C09015=1043.792,433.131,-138.600,175.491,44.902,159.085
C09016=1043.804,433.376,-138.650,175.504,44.911,159.089
C09017=1043.815,433.620,-138.700,175.518,44.920,159.093
C09018=1043.827,433.865,-138.751,175.531,44.929,159.097
C09019=1043.838,434.091,-138.798,175.543,44.937,159.100
C09020=1043.848,434.319,-138.844,175.556,44.945,159.104
C09021=1043.860,434.545,-138.891,175.568,44.954,159.108
C09022=1043.870,434.771,-138.938,175.581,44.962,159.111
C09023=1043.881,434.997,-138.985,175.594,44.970,159.115
C09024=1043.892,435.223,-139.032,175.606,44.979,159.118
C09025=1043.903,435.450,-139.079,175.619,44.987,159.122
C09026=1043.914,435.676,-139.126,175.632,44.995,159.126
C09027=1043.926,435.921,-139.177,175.646,45.005,159.130
C09028=1043.938,436.166,-139.228,175.660,45.013,159.134
C09029=1043.949,436.409,-139.279,175.674,45.023,159.138
C09030=1043.961,436.654,-139.330,175.687,45.032,159.142
C09031=1043.973,436.898,-139.382,175.702,45.041,159.146
C09032=1043.985,437.143,-139.433,175.715,45.050,159.150
C09033=1043.997,437.388,-139.485,175.730,45.059,159.154
C09034=1044.010,437.632,-139.535,175.743,45.069,159.158
C09035=1044.021,437.876,-139.587,175.758,45.078,159.162
C09036=1044.033,438.121,-139.638,175.773,45.087,159.166
C09037=1044.046,438.365,-139.690,175.787,45.097,159.170
C09038=1044.057,438.609,-139.742,175.801,45.106,159.174
C09039=1044.069,438.854,-139.793,175.815,45.116,159.179
C09040=1044.081,439.098,-139.845,175.830,45.125,159.183
C09041=1044.093,439.342,-139.897,175.845,45.135,159.187
C09042=1044.106,439.587,-139.949,175.860,45.144,159.191
C09043=1044.118,439.831,-140.001,175.874,45.154,159.196
C09044=1044.130,440.075,-140.053,175.888,45.163,159.200
C09045=1044.142,440.319,-140.105,175.903,45.173,159.204
C09046=1044.155,440.564,-140.157,175.918,45.183,159.208
C09047=1044.167,440.808,-140.209,175.933,45.192,159.213
C09048=1044.179,441.052,-140.261,175.948,45.202,159.217
C09049=1044.192,441.297,-140.313,175.963,45.212,159.222
C09050=1044.204,441.540,-140.365,175.978,45.221,159.226
C09051=1044.216,441.784,-140.418,175.993,45.231,159.230
C09052=1044.230,442.028,-140.471,176.009,45.241,159.235
C09053=1044.242,442.272,-140.523,176.024,45.251,159.239
C09054=1044.255,442.517,-140.575,176.039,45.261,159.244
C09055=1044.267,442.761,-140.627,176.054,45.271,159.248
C09056=1044.279,443.005,-140.681,176.070,45.280,159.253
C09057=1044.292,443.249,-140.734,176.086,45.291,159.257
C09058=1044.304,443.493,-140.787,176.101,45.301,159.262
C09059=1044.317,443.737,-140.839,176.116,45.311,159.266
C09060=1044.330,443.981,-140.892,176.133,45.321,159.271
C09061=1044.343,444.225,-140.945,176.148,45.331,159.275
C09062=1044.355,444.469,-140.998,176.164,45.341,159.280
C09063=1044.368,444.712,-141.050,176.180,45.351,159.285
C09064=1044.381,444.956,-141.104,176.196,45.361,159.289
C09065=1044.394,445.199,-141.157,176.212,45.371,159.294
C09066=1044.408,445.443,-141.210,176.228,45.382,159.299
C09067=1044.421,445.686,-141.262,176.244,45.392,159.303
C09068=1044.436,445.929,-141.313,176.260,45.401,159.308
C09069=1044.451,446.173,-141.365,176.277,45.411,159.312
C09070=1044.467,446.417,-141.415,176.293,45.420,159.317
C09071=1044.483,446.661,-141.466,176.309,45.430,159.321
C09072=1044.500,446.904,-141.516,176.325,45.439,159.326
C09073=1044.518,447.148,-141.565,176.343,45.449,159.331
C09074=1044.536,447.393,-141.614,176.359,45.458,159.335
C09075=1044.555,447.637,-141.662,176.376,45.467,159.339
C09076=1044.575,447.881,-141.710,176.392,45.476,159.344
C09077=1044.595,448.126,-141.756,176.409,45.485,159.348
C09078=1044.616,448.370,-141.804,176.426,45.493,159.353
C09079=1044.635,448.593,-141.846,176.442,45.501,159.357
C09080=1044.656,448.816,-141.888,176.457,45.509,159.361
C09081=1044.676,449.038,-141.929,176.473,45.517,159.365
C09082=1044.697,449.261,-141.970,176.489,45.524,159.368
C09083=1044.719,449.485,-142.011,176.505,45.531,159.372
C09084=1044.740,449.707,-142.051,176.520,45.539,159.376
C09085=1044.763,449.931,-142.090,176.537,45.546,159.380
C09086=1044.787,450.153,-142.130,176.553,45.553,159.384
C09087=1044.813,450.399,-142.172,176.569,45.561,159.388
C09088=1044.839,450.644,-142.215,176.588,45.568,159.392
C09089=1044.867,450.890,-142.256,176.606,45.576,159.397
C09090=1044.894,451.135,-142.298,176.623,45.583,159.401
C09091=1044.591,451.173,-142.608,176.625,45.666,159.425
C09092=1044.562,450.927,-142.567,176.608,45.658,159.421
C09093=1044.535,450.683,-142.525,176.589,45.651,159.417
C09094=1044.508,450.437,-142.483,176.571,45.644,159.413
C09095=1044.482,450.192,-142.441,176.554,45.636,159.409
C09096=1044.460,449.977,-142.403,176.539,45.629,159.405
C09097=1044.438,449.762,-142.365,176.523,45.622,159.401
C09098=1044.416,449.547,-142.327,176.507,45.615,159.397
C09099=1044.395,449.333,-142.287,176.492,45.608,159.394
C09100=1044.374,449.118,-142.248,176.477,45.601,159.390
C09101=1044.354,448.903,-142.208,176.462,45.594,159.386
C09102=1044.335,448.689,-142.168,176.447,45.586,159.382
C09103=1044.316,448.474,-142.127,176.432,45.580,159.379
C09104=1044.294,448.229,-142.081,176.415,45.571,159.374
C09105=1044.274,447.985,-142.034,176.397,45.562,159.370
C09106=1044.254,447.740,-141.987,176.381,45.554,159.365
C09107=1044.235,447.496,-141.939,176.364,45.544,159.361
C09108=1044.215,447.252,-141.890,176.347,45.535,159.356
C09109=1044.198,447.008,-141.841,176.331,45.526,159.352
C09110=1044.181,446.764,-141.791,176.314,45.517,159.347
C09111=1044.164,446.521,-141.742,176.297,45.508,159.343
C09112=1044.147,446.276,-141.691,176.281,45.498,159.338
C09113=1044.132,446.032,-141.640,176.265,45.489,159.334
C09114=1044.117,445.789,-141.589,176.248,45.479,159.329
C09115=1044.103,445.546,-141.537,176.232,45.469,159.325
C09116=1044.089,445.302,-141.485,176.216,45.459,159.320
C09117=1044.076,445.059,-141.431,176.200,45.449,159.315
C09118=1044.063,444.816,-141.378,176.183,45.439,159.311
C09119=1044.050,444.573,-141.326,176.168,45.429,159.306
C09120=1044.037,444.329,-141.273,176.152,45.419,159.301
C09121=1044.025,444.085,-141.219,176.136,45.409,159.297
C09122=1044.012,443.841,-141.167,176.121,45.399,159.292
C09123=1043.999,443.597,-141.114,176.104,45.389,159.288
C09124=1043.986,443.353,-141.061,176.089,45.379,159.283
C09125=1043.974,443.109,-141.008,176.074,45.369,159.278
C09126=1043.961,442.865,-140.955,176.058,45.360,159.274
C09127=1043.949,442.621,-140.903,176.042,45.349,159.269
C09128=1043.936,442.376,-140.851,176.027,45.339,159.265
C09129=1043.923,442.133,-140.798,176.012,45.330,159.261
C09130=1043.910,441.888,-140.745,175.997,45.320,159.256
C09131=1043.898,441.645,-140.693,175.982,45.310,159.252
C09132=1043.886,441.400,-140.640,175.966,45.300,159.247
C09133=1043.874,441.156,-140.588,175.951,45.290,159.243
C09134=1043.861,440.911,-140.535,175.936,45.281,159.239
C09135=1043.849,440.667,-140.483,175.921,45.271,159.234
C09136=1043.837,440.423,-140.431,175.906,45.262,159.230
C09137=1043.824,440.179,-140.379,175.891,45.252,159.226
C09138=1043.812,439.935,-140.328,175.876,45.243,159.221
C09139=1043.799,439.691,-140.276,175.861,45.233,159.217
C09140=1043.787,439.447,-140.224,175.846,45.224,159.213
C09141=1043.775,439.202,-140.172,175.832,45.215,159.209
C09142=1043.762,438.958,-140.120,175.818,45.205,159.204
C09143=1043.751,438.713,-140.068,175.803,45.195,159.200
C09144=1043.738,438.469,-140.016,175.788,45.186,159.196
C09145=1043.727,438.225,-139.965,175.773,45.177,159.192
C09146=1043.715,437.980,-139.913,175.760,45.168,159.188
C09147=1043.702,437.736,-139.861,175.745,45.158,159.184
C09148=1043.691,437.492,-139.810,175.731,45.149,159.179
C09149=1043.679,437.247,-139.759,175.717,45.140,159.175
C09150=1043.666,437.003,-139.708,175.702,45.131,159.171
C09151=1043.654,436.759,-139.656,175.688,45.121,159.167
C09152=1043.642,436.514,-139.605,175.675,45.112,159.163
C09153=1043.631,436.270,-139.554,175.660,45.103,159.159
C09154=1043.619,436.025,-139.503,175.647,45.094,159.155
C09155=1043.608,435.781,-139.452,175.633,45.085,159.151
C09156=1043.596,435.554,-139.405,175.619,45.077,159.148
C09157=1043.585,435.326,-139.358,175.607,45.068,159.144
C09158=1043.574,435.099,-139.310,175.594,45.060,159.140
C09159=1043.562,434.872,-139.263,175.581,45.052,159.137
C09160=1043.552,434.645,-139.216,175.568,45.044,159.133
C09161=1043.541,434.417,-139.169,175.556,45.035,159.129
C09162=1043.530,434.190,-139.122,175.543,45.027,159.126
C09163=1043.519,433.963,-139.075,175.530,45.019,159.122
C09164=1043.508,433.718,-139.024,175.517,45.010,159.118
C09165=1043.495,433.473,-138.974,175.504,45.001,159.115
C09166=1043.484,433.229,-138.923,175.491,44.993,159.111
C09167=1043.472,432.984,-138.873,175.477,44.984,159.107
C09168=1043.461,432.740,-138.823,175.464,44.975,159.103
C09169=1043.449,432.495,-138.772,175.451,44.967,159.099
C09170=1043.438,432.250,-138.722,175.438,44.958,159.096
C09171=1043.427,432.006,-138.672,175.425,44.949,159.092
C09172=1043.414,431.761,-138.622,175.412,44.941,159.088
C09173=1043.404,431.516,-138.572,175.399,44.932,159.084
C09174=1043.392,431.271,-138.522,175.386,44.924,159.081
C09175=1043.380,431.027,-138.472,175.372,44.915,159.077
C09176=1043.370,430.782,-138.422,175.359,44.907,159.073
C09177=1043.358,430.538,-138.372,175.347,44.898,159.070
C09178=1043.346,430.293,-138.322,175.334,44.890,159.066
C09179=1043.336,430.047,-138.272,175.322,44.881,159.063
C09180=1043.324,429.803,-138.222,175.309,44.873,159.059
C09181=1043.313,429.558,-138.173,175.296,44.864,159.055
C09182=1043.302,429.314,-138.124,175.283,44.856,159.052
C09183=1043.291,429.069,-138.073,175.271,44.848,159.048
C09184=1043.280,428.823,-138.024,175.258,44.840,159.045
C09185=1043.268,428.579,-137.974,175.245,44.831,159.041
C09186=1043.257,428.334,-137.925,175.234,44.823,159.038
C09187=1043.246,428.089,-137.876,175.221,44.815,159.034
C09188=1043.235,427.844,-137.827,175.208,44.807,159.031
C09189=1043.224,427.599,-137.777,175.196,44.799,159.027
C09190=1043.213,427.354,-137.728,175.184,44.791,159.024
C09191=1043.201,427.110,-137.679,175.172,44.782,159.020
C09192=1043.191,426.865,-137.630,175.159,44.774,159.017
C09193=1043.180,426.619,-137.581,175.148,44.766,159.014
C09194=1043.168,426.374,-137.532,175.135,44.758,159.010
C09195=1043.158,426.129,-137.483,175.123,44.750,159.007
C09196=1043.147,425.885,-137.435,175.111,44.742,159.003
C09197=1043.136,425.640,-137.386,175.099,44.734,159.000
C09198=1043.125,425.395,-137.336,175.087,44.726,158.997
C09199=1043.114,425.150,-137.288,175.075,44.719,158.993
C09200=1043.103,424.906,-137.239,175.063,44.710,158.990
C09201=1043.092,424.660,-137.191,175.051,44.703,158.987
C09202=1043.082,424.414,-137.142,175.040,44.695,158.983
C09203=1043.070,424.169,-137.094,175.028,44.687,158.980
C09204=1043.060,423.925,-137.045,175.017,44.679,158.977
C09205=1043.049,423.680,-136.997,175.004,44.671,158.974
C09206=1043.037,423.434,-136.948,174.993,44.664,158.970
C09207=1043.027,423.190,-136.901,174.981,44.656,158.967
C09208=1043.016,422.944,-136.852,174.970,44.648,158.964
C09209=1043.005,422.700,-136.804,174.959,44.641,158.961
C09210=1042.995,422.454,-136.755,174.946,44.633,158.957
C09211=1042.984,422.209,-136.707,174.935,44.626,158.954
C09212=1042.974,421.963,-136.660,174.924,44.618,158.951
C09213=1042.963,421.718,-136.612,174.913,44.610,158.948
C09214=1042.952,421.473,-136.564,174.901,44.602,158.945
C09215=1042.942,421.229,-136.516,174.890,44.595,158.942
C09216=1042.933,421.011,-136.474,174.881,44.589,158.939
C09217=1042.922,420.793,-136.431,174.870,44.582,158.936
C09218=1042.913,420.575,-136.388,174.860,44.575,158.934
C09219=1042.904,420.358,-136.346,174.850,44.568,158.931
C09220=1042.894,420.140,-136.304,174.841,44.562,158.928
C09221=1042.885,419.922,-136.261,174.831,44.555,158.925
C09222=1042.876,419.704,-136.219,174.821,44.549,158.923
C09223=1042.866,419.487,-136.177,174.811,44.542,158.920
C09224=1042.856,419.242,-136.129,174.800,44.535,158.917
C09225=1042.846,418.997,-136.082,174.790,44.528,158.914
C09226=1042.835,418.752,-136.034,174.778,44.520,158.911
C09227=1042.825,418.507,-135.987,174.767,44.513,158.908
C09228=1042.815,418.260,-135.939,174.756,44.506,158.905
C09229=1042.804,418.015,-135.892,174.745,44.499,158.902
C09230=1042.794,417.770,-135.845,174.735,44.491,158.899
C09231=1042.784,417.525,-135.798,174.724,44.484,158.896
C09232=1042.774,417.279,-135.751,174.713,44.477,158.893
C09233=1042.764,417.034,-135.703,174.703,44.470,158.890
C09234=1042.752,416.789,-135.656,174.692,44.462,158.887
C09235=1042.742,416.543,-135.609,174.682,44.456,158.884
C09236=1042.732,416.297,-135.563,174.671,44.449,158.881
C09237=1042.722,416.052,-135.515,174.661,44.442,158.879
C09238=1042.712,415.807,-135.468,174.650,44.434,158.876
C09239=1042.701,415.561,-135.422,174.639,44.427,158.873
C09240=1042.691,415.317,-135.375,174.629,44.420,158.870
C09241=1042.681,415.071,-135.328,174.618,44.413,158.867
C09242=1042.671,414.825,-135.282,174.609,44.406,158.864
C09243=1042.660,414.580,-135.235,174.598,44.399,158.861
C09244=1042.650,414.335,-135.189,174.588,44.393,158.859
C09245=1042.640,414.089,-135.141,174.577,44.386,158.856
C09246=1042.630,413.843,-135.095,174.568,44.379,158.853
C09247=1042.620,413.598,-135.049,174.557,44.372,158.850
C09248=1042.610,413.353,-135.002,174.547,44.365,158.848
C09249=1042.600,413.107,-134.956,174.537,44.358,158.845
C09250=1042.590,412.861,-134.909,174.527,44.351,158.842
C09251=1042.580,412.616,-134.864,174.516,44.345,158.839
C09252=1042.571,412.371,-134.817,174.506,44.338,158.836
C09253=1042.560,412.125,-134.770,174.497,44.331,158.834
C09254=1042.551,411.880,-134.724,174.486,44.325,158.831
C09255=1042.541,411.634,-134.679,174.477,44.318,158.828
C09256=1042.530,411.388,-134.633,174.466,44.311,158.826
C09257=1042.521,411.143,-134.586,174.457,44.305,158.823
C09258=1042.510,410.897,-134.541,174.447,44.298,158.820
C09259=1042.500,410.652,-134.494,174.436,44.292,158.818
C09260=1042.490,410.407,-134.449,174.427,44.285,158.815
C09261=1042.481,410.160,-134.403,174.417,44.278,158.813
C09262=1042.471,409.915,-134.357,174.408,44.272,158.810
C09263=1042.460,409.670,-134.311,174.397,44.265,158.807
C09264=1042.451,409.424,-134.266,174.388,44.259,158.805
C09265=1042.440,409.178,-134.220,174.378,44.252,158.802
C09266=1042.431,408.932,-134.175,174.369,44.246,158.800
C09267=1042.421,408.688,-134.129,174.360,44.239,158.797
C09268=1042.412,408.441,-134.083,174.349,44.233,158.794
C09269=1042.402,408.196,-134.038,174.340,44.227,158.792
C09270=1042.392,407.950,-133.993,174.330,44.220,158.789
C09271=1042.383,407.704,-133.947,174.321,44.214,158.787
C09272=1042.373,407.459,-133.902,174.312,44.207,158.784
C09273=1042.364,407.213,-133.856,174.302,44.201,158.782
C09274=1042.353,406.967,-133.811,174.293,44.195,158.779
C09275=1042.344,406.722,-133.766,174.284,44.189,158.777
C09276=1042.336,406.508,-133.727,174.275,44.183,158.774
C09277=1042.327,406.295,-133.687,174.267,44.178,158.772
C09278=1042.319,406.081,-133.648,174.259,44.172,158.770
C09279=1042.310,405.867,-133.608,174.251,44.167,158.768
C09280=1042.302,405.654,-133.569,174.242,44.161,158.766
C09281=1042.293,405.440,-133.530,174.235,44.156,158.764
C09282=1042.285,405.227,-133.490,174.227,44.150,158.762
C09283=1042.278,405.013,-133.452,174.219,44.145,158.759
C09284=1042.268,404.767,-133.407,174.210,44.139,158.757
C09285=1042.258,404.522,-133.362,174.200,44.133,158.755
C09286=1042.249,404.276,-133.317,174.191,44.127,158.752
C09287=1042.240,404.030,-133.272,174.182,44.121,158.750
C09288=1042.230,403.784,-133.228,174.173,44.115,158.747
C09289=1042.221,403.538,-133.182,174.164,44.109,158.745
C09290=1042.211,403.292,-133.137,174.155,44.102,158.743
C09291=1042.201,403.046,-133.093,174.146,44.097,158.740
C09292=1042.192,402.801,-133.048,174.137,44.090,158.738
C09293=1042.183,402.555,-133.003,174.128,44.084,158.735
C09294=1042.174,402.309,-132.959,174.119,44.079,158.733
C09295=1042.164,402.064,-132.914,174.110,44.073,158.731
C09296=1042.155,401.818,-132.870,174.102,44.067,158.729
C09297=1042.145,401.572,-132.826,174.093,44.061,158.726
C09298=1042.136,401.326,-132.781,174.084,44.055,158.724
C09299=1042.126,401.080,-132.737,174.075,44.049,158.721
C09300=1042.118,400.834,-132.693,174.067,44.043,158.719
C09301=1042.108,400.589,-132.648,174.058,44.037,158.717
C09302=1042.099,400.343,-132.604,174.049,44.031,158.715
C09303=1042.090,400.096,-132.560,174.040,44.026,158.712
C09304=1042.080,399.851,-132.516,174.032,44.020,158.710
C09305=1042.071,399.605,-132.472,174.023,44.014,158.708
C09306=1042.061,399.359,-132.428,174.014,44.009,158.706
C09307=1042.052,399.113,-132.384,174.006,44.003,158.703
C09308=1042.043,398.867,-132.340,173.997,43.997,158.701
C09309=1042.034,398.621,-132.296,173.988,43.992,158.699
C09310=1042.024,398.375,-132.252,173.980,43.986,158.697
C09311=1042.016,398.130,-132.208,173.971,43.980,158.695
C09312=1042.006,397.884,-132.164,173.962,43.974,158.692
C09313=1041.997,397.638,-132.121,173.954,43.969,158.690
C09314=1041.988,397.392,-132.076,173.945,43.963,158.688
C09315=1041.979,397.147,-132.033,173.938,43.957,158.686
C09316=1041.969,396.900,-131.990,173.929,43.952,158.684
C09317=1041.960,396.655,-131.946,173.921,43.946,158.681
C09318=1041.951,396.409,-131.902,173.912,43.941,158.679
C09319=1041.943,396.163,-131.859,173.904,43.935,158.677
C09320=1041.933,395.916,-131.815,173.895,43.930,158.675
C09321=1041.924,395.671,-131.771,173.888,43.924,158.673
C09322=1041.915,395.424,-131.728,173.879,43.919,158.671
C09323=1041.906,395.179,-131.685,173.871,43.913,158.669
C09324=1041.897,394.933,-131.642,173.862,43.908,158.666
C09325=1041.888,394.686,-131.598,173.855,43.902,158.664
C09326=1041.879,394.441,-131.554,173.846,43.897,158.662
C09327=1041.869,394.194,-131.512,173.838,43.892,158.660
C09328=1041.861,393.948,-131.469,173.829,43.886,158.658
C09329=1041.852,393.703,-131.425,173.822,43.881,158.656
C09330=1041.842,393.456,-131.382,173.813,43.875,158.654
C09331=1041.834,393.210,-131.339,173.805,43.870,158.652
C09332=1041.825,392.964,-131.296,173.798,43.865,158.650
C09333=1041.816,392.719,-131.253,173.789,43.860,158.648
C09334=1041.807,392.472,-131.209,173.781,43.854,158.646
C09335=1041.798,392.226,-131.166,173.774,43.849,158.644
C09336=1041.783,391.818,-131.096,173.760,43.840,158.640
C09337=1041.769,391.411,-131.025,173.747,43.831,158.637
C09338=1041.754,391.003,-130.954,173.733,43.823,158.634
C09339=1041.739,390.595,-130.883,173.720,43.814,158.630
C09340=1041.731,390.349,-130.840,173.713,43.809,158.628
C09341=1041.722,390.103,-130.798,173.705,43.804,158.627
C09342=1041.713,389.857,-130.755,173.697,43.799,158.624
C09343=1041.704,389.610,-130.713,173.689,43.794,158.622
C09344=1041.695,389.364,-130.670,173.681,43.789,158.621
C09345=1041.686,389.119,-130.627,173.674,43.784,158.619
C09346=1041.678,388.872,-130.585,173.666,43.778,158.617
C09347=1041.668,388.626,-130.543,173.658,43.774,158.615
C09348=1041.660,388.379,-130.500,173.650,43.768,158.613
C09349=1041.651,388.134,-130.458,173.643,43.764,158.611
C09350=1041.643,387.887,-130.416,173.635,43.759,158.609
C09351=1041.634,387.641,-130.373,173.628,43.753,158.607
C09352=1041.625,387.395,-130.331,173.619,43.749,158.605
C09353=1041.616,387.148,-130.289,173.612,43.744,158.603
C09354=1041.607,386.902,-130.247,173.604,43.739,158.601
C09355=1041.598,386.656,-130.205,173.597,43.734,158.600
C09356=1041.589,386.410,-130.163,173.590,43.729,158.598
C09357=1041.581,386.164,-130.120,173.582,43.724,158.596
C09358=1041.572,385.918,-130.079,173.575,43.720,158.594
C09359=1041.564,385.672,-130.037,173.566,43.714,158.592
C09360=1041.555,385.425,-129.995,173.559,43.710,158.590
C09361=1041.546,385.179,-129.953,173.552,43.705,158.588
C09362=1041.537,384.932,-129.911,173.544,43.700,158.587
C09363=1041.529,384.686,-129.870,173.537,43.695,158.585
C09364=1041.520,384.440,-129.828,173.530,43.690,158.583
C09365=1041.512,384.194,-129.786,173.522,43.686,158.581
C09366=1041.503,383.947,-129.744,173.515,43.681,158.579
C09367=1041.494,383.701,-129.703,173.508,43.677,158.578
C09368=1041.486,383.455,-129.661,173.500,43.672,158.576
C09369=1041.477,383.209,-129.620,173.493,43.667,158.574
C09370=1041.469,382.962,-129.577,173.486,43.662,158.572
C09371=1041.460,382.716,-129.536,173.478,43.657,158.570
C09372=1041.452,382.469,-129.495,173.471,43.652,158.568
C09373=1041.443,382.223,-129.453,173.464,43.648,158.567
C09374=1041.435,381.977,-129.411,173.456,43.643,158.565
C09375=1041.426,381.731,-129.369,173.449,43.639,158.563
C09376=1041.418,381.484,-129.328,173.442,43.634,158.561
C09377=1041.409,381.238,-129.287,173.435,43.630,158.560
C09378=1041.400,380.992,-129.245,173.427,43.625,158.558
C09379=1041.393,380.745,-129.204,173.421,43.620,158.556
C09380=1041.384,380.499,-129.162,173.414,43.615,158.554
C09381=1041.376,380.253,-129.122,173.407,43.611,158.553
C09382=1041.367,380.006,-129.080,173.399,43.606,158.551
C09383=1041.359,379.760,-129.039,173.392,43.602,158.549
C09384=1041.347,379.392,-128.977,173.382,43.595,158.547
C09385=1041.334,379.025,-128.916,173.372,43.588,158.544
C09386=1041.322,378.657,-128.854,173.360,43.582,158.542
C09387=1041.309,378.290,-128.794,173.350,43.575,158.539
C09388=1041.300,378.043,-128.753,173.343,43.571,158.537
C09389=1041.292,377.797,-128.712,173.337,43.566,158.536
C09390=1041.284,377.551,-128.672,173.330,43.562,158.534
C09391=1041.275,377.304,-128.630,173.323,43.558,158.533
C09392=1041.267,377.051,-128.589,173.315,43.553,158.531
C09393=1041.259,376.798,-128.547,173.308,43.549,158.529
C09394=1041.250,376.546,-128.505,173.301,43.544,158.527
C09395=1041.241,376.293,-128.463,173.294,43.540,158.526
C09396=1041.233,376.046,-128.423,173.288,43.535,158.524
C09397=1041.224,375.799,-128.382,173.281,43.531,158.523
C09398=1041.216,375.553,-128.341,173.274,43.527,158.521
C09399=1041.208,375.307,-128.300,173.267,43.523,158.519
C09400=1041.200,375.060,-128.260,173.261,43.518,158.518
C09401=1041.192,374.813,-128.219,173.254,43.514,158.516
C09402=1041.183,374.567,-128.179,173.246,43.510,158.514
C09403=1041.175,374.321,-128.139,173.240,43.505,158.513
C09404=1041.167,374.074,-128.098,173.233,43.502,158.511
C09405=1041.159,373.827,-128.058,173.226,43.497,158.510
C09406=1041.151,373.581,-128.017,173.220,43.493,158.508
C09407=1041.143,373.334,-127.977,173.213,43.488,158.506
C09408=1041.134,373.088,-127.937,173.206,43.485,158.505
C09409=1041.126,372.841,-127.897,173.200,43.480,158.503
C09410=1041.117,372.594,-127.856,173.193,43.476,158.502
C09411=1041.110,372.347,-127.816,173.186,43.472,158.500
C09412=1041.102,372.101,-127.775,173.180,43.468,158.499
C09413=1041.094,371.854,-127.735,173.173,43.463,158.497
C09414=1041.085,371.608,-127.695,173.167,43.459,158.496
C09415=1041.077,371.361,-127.655,173.160,43.455,158.494
C09416=1041.069,371.115,-127.615,173.153,43.451,158.492
C09417=1041.062,370.868,-127.575,173.147,43.447,158.491
C09418=1041.054,370.622,-127.534,173.141,43.443,158.489
C09419=1041.045,370.375,-127.495,173.134,43.439,158.488
C09420=1041.038,370.128,-127.455,173.128,43.435,158.486
C09421=1041.029,369.882,-127.415,173.122,43.431,158.485
C09422=1041.021,369.636,-127.375,173.115,43.427,158.483
C09423=1041.013,369.389,-127.335,173.108,43.423,158.482
C09424=1041.004,369.141,-127.295,173.102,43.419,158.480
C09425=1040.996,368.895,-127.256,173.095,43.415,158.479
C09426=1040.988,368.648,-127.216,173.089,43.411,158.477
C09427=1040.980,368.403,-127.176,173.082,43.408,158.476
C09428=1040.972,368.156,-127.136,173.076,43.403,158.474
C09429=1040.964,367.909,-127.097,173.070,43.399,158.473
C09430=1040.956,367.662,-127.057,173.064,43.395,158.471
C09431=1040.948,367.416,-127.018,173.057,43.392,158.470
C09432=1040.940,367.169,-126.978,173.051,43.388,158.469
C09433=1040.931,366.922,-126.939,173.044,43.384,158.467
C09434=1040.924,366.675,-126.899,173.038,43.380,158.466
C09435=1040.916,366.428,-126.860,173.033,43.376,158.464
C09436=1040.908,366.181,-126.820,173.026,43.372,158.463
C09437=1040.899,365.934,-126.781,173.020,43.368,158.461
C09438=1040.892,365.688,-126.741,173.013,43.365,158.460
C09439=1040.884,365.442,-126.702,173.007,43.361,158.458
C09440=1040.876,365.194,-126.663,173.000,43.357,158.457
C09441=1040.868,364.948,-126.623,172.995,43.353,158.456
C09442=1040.860,364.701,-126.583,172.989,43.350,158.454
C09443=1040.852,364.455,-126.545,172.982,43.346,158.453
C09444=1040.844,364.208,-126.506,172.976,43.342,158.451
C09445=1040.836,363.961,-126.466,172.970,43.338,158.450
C09446=1040.828,363.714,-126.427,172.964,43.334,158.448
C09447=1040.821,363.467,-126.388,172.958,43.331,158.447
C09448=1040.809,363.113,-126.331,172.950,43.325,158.445
C09449=1040.799,362.759,-126.275,172.940,43.320,158.443
C09450=1040.788,362.405,-126.219,172.932,43.315,158.441
C09451=1040.776,362.051,-126.164,172.923,43.309,158.439
C09452=1040.769,361.804,-126.124,172.917,43.305,158.438
C09453=1040.760,361.557,-126.085,172.911,43.302,158.437
C09454=1040.753,361.311,-126.047,172.905,43.298,158.435
C09455=1040.744,361.064,-126.008,172.899,43.295,158.434
C09456=1040.736,360.816,-125.970,172.892,43.291,158.432
C09457=1040.729,360.570,-125.930,172.887,43.288,158.431
C09458=1040.721,360.323,-125.891,172.881,43.284,158.430
C09459=1040.713,360.076,-125.853,172.875,43.280,158.428
C09460=1040.705,359.829,-125.815,172.869,43.277,158.427
C09461=1040.697,359.582,-125.776,172.863,43.273,158.426
C09462=1040.689,359.336,-125.737,172.857,43.270,158.425
C09463=1040.682,359.089,-125.698,172.851,43.266,158.423
C09464=1040.674,358.842,-125.660,172.845,43.263,158.422
C09465=1040.666,358.595,-125.621,172.840,43.259,158.421
C09466=1040.659,358.348,-125.583,172.834,43.256,158.419
C09467=1040.650,358.101,-125.544,172.828,43.252,158.418
C09468=1040.643,357.855,-125.506,172.822,43.249,158.417
C09469=1040.635,357.607,-125.467,172.816,43.245,158.415
C09470=1040.627,357.361,-125.429,172.810,43.242,158.414
C09471=1040.620,357.113,-125.390,172.805,43.238,158.413
C09472=1040.612,356.867,-125.352,172.799,43.234,158.411
C09473=1040.604,356.619,-125.314,172.792,43.231,158.410
C09474=1040.597,356.372,-125.275,172.787,43.228,158.409
C09475=1040.589,356.126,-125.237,172.781,43.224,158.408
C09476=1040.581,355.879,-125.199,172.776,43.221,158.406
C09477=1040.574,355.632,-125.160,172.770,43.218,158.405
C09478=1040.566,355.384,-125.122,172.765,43.214,158.404
C09479=1040.558,355.138,-125.084,172.758,43.211,158.403
C09480=1040.549,354.891,-125.046,172.752,43.208,158.401
C09481=1040.542,354.644,-125.009,172.747,43.204,158.400
C09482=1040.535,354.397,-124.970,172.741,43.201,158.399
C09483=1040.527,354.149,-124.932,172.736,43.198,158.398
C09484=1040.519,353.903,-124.894,172.730,43.194,158.396
C09485=1040.512,353.656,-124.856,172.725,43.191,158.395
C09486=1040.504,353.409,-124.818,172.718,43.188,158.394
C09487=1040.496,353.162,-124.780,172.713,43.184,158.393
C09488=1040.489,352.915,-124.742,172.707,43.181,158.391
C09489=1040.481,352.668,-124.704,172.702,43.178,158.390
C09490=1040.474,352.421,-124.666,172.696,43.175,158.389
C09491=1040.466,352.174,-124.629,172.691,43.171,158.388
C09492=1040.458,351.927,-124.591,172.685,43.168,158.387
C09493=1040.451,351.680,-124.553,172.680,43.165,158.385
C09494=1040.443,351.433,-124.515,172.674,43.162,158.384
C09495=1040.435,351.186,-124.477,172.669,43.158,158.383
C09496=1040.428,350.939,-124.440,172.663,43.155,158.382
C09497=1040.421,350.692,-124.402,172.658,43.152,158.381
C09498=1040.413,350.445,-124.364,172.652,43.149,158.379
C09499=1040.405,350.198,-124.327,172.647,43.146,158.378
C09500=1040.397,349.950,-124.289,172.641,43.142,158.377
C09501=1040.390,349.703,-124.252,172.636,43.139,158.376
C09502=1040.383,349.457,-124.213,172.630,43.136,158.375
C09503=1040.375,349.210,-124.177,172.625,43.133,158.373
C09504=1040.364,348.861,-124.124,172.617,43.128,158.372
C09505=1040.354,348.514,-124.071,172.609,43.124,158.370
C09506=1040.342,348.165,-124.019,172.602,43.120,158.369
C09507=1040.332,347.817,-123.966,172.594,43.115,158.367
C09508=1040.324,347.570,-123.929,172.588,43.112,158.366
C09509=1040.317,347.323,-123.891,172.583,43.109,158.365
C09510=1040.310,347.076,-123.854,172.577,43.106,158.364
C09511=1040.302,346.829,-123.817,172.572,43.103,158.362
C09512=1040.295,346.581,-123.780,172.566,43.100,158.361
C09513=1040.288,346.334,-123.742,172.562,43.097,158.360
C09514=1040.280,346.087,-123.705,172.557,43.094,158.359
C09515=1040.273,345.840,-123.668,172.551,43.091,158.358
C09516=1040.265,345.594,-123.631,172.546,43.088,158.357
C09517=1040.258,345.346,-123.594,172.541,43.085,158.356
C09518=1040.250,345.099,-123.557,172.535,43.082,158.355
C09519=1040.242,344.852,-123.520,172.530,43.079,158.354
C09520=1040.235,344.605,-123.482,172.524,43.076,158.352
C09521=1040.228,344.357,-123.446,172.519,43.073,158.351
C09522=1040.220,344.110,-123.408,172.514,43.070,158.350
C09523=1040.212,343.863,-123.371,172.508,43.067,158.349
C09524=1040.205,343.616,-123.335,172.504,43.064,158.348
C09525=1040.197,343.369,-123.298,172.499,43.061,158.347
C09526=1040.190,343.121,-123.261,172.493,43.058,158.346
C09527=1040.183,342.875,-123.224,172.488,43.055,158.345
C09528=1040.176,342.627,-123.187,172.483,43.052,158.343
C09529=1040.168,342.380,-123.151,172.477,43.049,158.342
C09530=1040.161,342.132,-123.114,172.473,43.046,158.341
C09531=1040.153,341.886,-123.077,172.468,43.043,158.340
C09532=1040.146,341.638,-123.040,172.462,43.040,158.339
C09533=1040.138,341.391,-123.003,172.457,43.038,158.338
C09534=1040.131,341.144,-122.967,172.452,43.035,158.337
C09535=1040.124,340.897,-122.930,172.446,43.032,158.336
C09536=1040.116,340.650,-122.893,172.442,43.029,158.335
C09537=1040.109,340.402,-122.857,172.437,43.026,158.334
C09538=1040.102,340.155,-122.820,172.431,43.024,158.333
C09539=1040.095,339.908,-122.785,172.426,43.021,158.332
C09540=1040.087,339.661,-122.748,172.421,43.018,158.331
C09541=1040.079,339.414,-122.711,172.417,43.015,158.330
C09542=1040.072,339.166,-122.675,172.411,43.013,158.329
C09543=1040.064,338.918,-122.638,172.406,43.010,158.328
C09544=1040.057,338.672,-122.603,172.401,43.007,158.327
C09545=1040.049,338.425,-122.566,172.396,43.004,158.326
C09546=1040.042,338.177,-122.529,172.391,43.001,158.325
C09547=1040.035,337.930,-122.493,172.386,42.999,158.324
C09548=1040.028,337.683,-122.457,172.381,42.996,158.322
C09549=1040.021,337.435,-122.420,172.376,42.993,158.322
C09550=1040.014,337.188,-122.384,172.371,42.990,158.321
C09551=1040.006,336.941,-122.348,172.366,42.987,158.319
C09552=1039.998,336.693,-122.312,172.361,42.985,158.319
C09553=1039.992,336.446,-122.275,172.357,42.982,158.317
C09554=1039.984,336.199,-122.239,172.351,42.979,158.316
C09555=1039.977,335.951,-122.203,172.346,42.977,158.316
C09556=1039.969,335.705,-122.167,172.341,42.974,158.314
C09557=1039.962,335.457,-122.131,172.337,42.972,158.314
C09558=1039.955,335.210,-122.094,172.331,42.969,158.312
C09559=1039.948,334.962,-122.059,172.326,42.966,158.311
C09560=1039.937,334.611,-122.008,172.320,42.962,158.310
C09561=1039.927,334.259,-121.957,172.313,42.959,158.309
C09562=1039.917,333.907,-121.906,172.306,42.955,158.307
C09563=1039.907,333.555,-121.855,172.298,42.952,158.306
C09564=1039.899,333.308,-121.818,172.294,42.948,158.305
C09565=1039.892,333.061,-121.783,172.289,42.946,158.304
C09566=1039.885,332.813,-121.747,172.284,42.943,158.303
C09567=1039.877,332.566,-121.711,172.280,42.941,158.302
C09568=1039.869,332.319,-121.676,172.275,42.938,158.301
C09569=1039.862,332.072,-121.640,172.269,42.936,158.300
C09570=1039.855,331.824,-121.604,172.265,42.933,158.299
C09571=1039.848,331.577,-121.569,172.260,42.931,158.298
C09572=1039.840,331.330,-121.533,172.256,42.928,158.297
C09573=1039.833,331.082,-121.498,172.251,42.925,158.296
C09574=1039.826,330.835,-121.462,172.246,42.923,158.295
C09575=1039.819,330.587,-121.426,172.241,42.920,158.294
C09576=1039.812,330.341,-121.391,172.236,42.918,158.293
C09577=1039.804,330.093,-121.355,172.232,42.915,158.293
C09578=1039.797,329.846,-121.319,172.227,42.913,158.292
C09579=1039.790,329.598,-121.284,172.222,42.910,158.291
C09580=1039.783,329.350,-121.249,172.218,42.908,158.290
C09581=1039.776,329.104,-121.213,172.213,42.905,158.289
C09582=1039.769,328.856,-121.177,172.208,42.903,158.288
C09583=1039.762,328.608,-121.142,172.203,42.900,158.287
C09584=1039.754,328.361,-121.106,172.198,42.898,158.286
C09585=1039.747,328.114,-121.071,172.194,42.896,158.285
C09586=1039.740,327.866,-121.036,172.189,42.893,158.284
C09587=1039.732,327.619,-121.001,172.185,42.891,158.283
C09588=1039.725,327.371,-120.966,172.180,42.889,158.283
C09589=1039.717,327.123,-120.931,172.175,42.886,158.282
C09590=1039.710,326.876,-120.896,172.171,42.884,158.281
C09591=1039.703,326.629,-120.862,172.166,42.881,158.280
C09592=1039.695,326.382,-120.825,172.162,42.879,158.279
C09593=1039.688,326.135,-120.791,172.156,42.877,158.278
C09594=1039.681,325.887,-120.756,172.152,42.874,158.277
C09595=1039.674,325.639,-120.720,172.147,42.872,158.276
C09596=1039.666,325.392,-120.686,172.143,42.869,158.275
C09597=1039.659,325.145,-120.651,172.138,42.867,158.274
C09598=1039.652,324.898,-120.616,172.134,42.865,158.274
C09599=1039.645,324.649,-120.581,172.129,42.863,158.273
C09600=1039.637,324.402,-120.547,172.125,42.860,158.272
C09601=1039.630,324.155,-120.512,172.120,42.858,158.271
C09602=1039.623,323.908,-120.477,172.115,42.856,158.270
C09603=1039.616,323.659,-120.441,172.111,42.853,158.269
C09604=1039.608,323.412,-120.407,172.107,42.851,158.268
C09605=1039.601,323.165,-120.372,172.102,42.849,158.268
C09606=1039.594,322.918,-120.337,172.098,42.846,158.267
C09607=1039.587,322.670,-120.303,172.093,42.844,158.266
C09608=1039.580,322.422,-120.267,172.089,42.842,158.265
C09609=1039.572,322.175,-120.233,172.084,42.839,158.264
C09610=1039.566,321.928,-120.198,172.080,42.837,158.263
C09611=1039.558,321.680,-120.164,172.075,42.835,158.262
C09612=1039.552,321.432,-120.129,172.070,42.833,158.262
C09613=1039.544,321.185,-120.094,172.065,42.830,158.261
C09614=1039.538,320.937,-120.060,172.062,42.828,158.260
C09615=1039.530,320.690,-120.025,172.056,42.826,158.259
C09616=1039.520,320.333,-119.975,172.051,42.823,158.258
C09617=1039.509,319.977,-119.926,172.045,42.820,158.257
C09618=1039.499,319.621,-119.875,172.038,42.816,158.255
C09619=1039.489,319.264,-119.825,172.032,42.813,158.254
C09620=1039.482,319.017,-119.791,172.027,42.811,158.253
C09621=1039.475,318.769,-119.756,172.023,42.809,158.253
C09622=1039.468,318.522,-119.722,172.019,42.806,158.252
C09623=1039.461,318.274,-119.687,172.014,42.805,158.251
C09624=1039.454,318.027,-119.653,172.010,42.802,158.250
C09625=1039.447,317.779,-119.618,172.005,42.800,158.249
C09626=1039.440,317.532,-119.584,172.001,42.798,158.248
C09627=1039.433,317.284,-119.549,171.997,42.795,158.248
C09628=1039.426,317.036,-119.515,171.992,42.794,158.247
C09629=1039.420,316.788,-119.481,171.988,42.791,158.246
C09630=1039.413,316.542,-119.447,171.984,42.789,158.245
C09631=1039.406,316.294,-119.413,171.979,42.787,158.244
C09632=1039.399,316.047,-119.378,171.975,42.784,158.243
C09633=1039.392,315.799,-119.344,171.971,42.782,158.243
C09634=1039.385,315.551,-119.310,171.966,42.780,158.242
C09635=1039.378,315.304,-119.275,171.962,42.778,158.241
C09636=1039.371,315.056,-119.241,171.958,42.776,158.240
C09637=1039.364,314.809,-119.207,171.953,42.774,158.239
C09638=1039.358,314.562,-119.172,171.949,42.771,158.239
C09639=1039.351,314.314,-119.138,171.945,42.769,158.238
C09640=1039.344,314.066,-119.104,171.941,42.767,158.237
C09641=1039.337,313.819,-119.070,171.936,42.765,158.236
C09642=1039.330,313.571,-119.036,171.932,42.763,158.235
C09643=1039.324,313.324,-119.001,171.928,42.761,158.235
C09644=1039.316,313.077,-118.968,171.923,42.759,158.234
C09645=1039.310,312.829,-118.933,171.919,42.756,158.233
C09646=1039.303,312.581,-118.899,171.915,42.755,158.232
C09647=1039.297,312.334,-118.865,171.911,42.752,158.231
C09648=1039.290,312.086,-118.831,171.906,42.750,158.231
C09649=1039.282,311.838,-118.798,171.903,42.748,158.230
C09650=1039.275,311.591,-118.764,171.899,42.746,158.229
C09651=1039.268,311.343,-118.730,171.894,42.744,158.228
C09652=1039.261,311.095,-118.696,171.890,42.742,158.228
C09653=1039.253,310.849,-118.663,171.886,42.740,158.227
C09654=1039.246,310.601,-118.629,171.882,42.738,158.226
C09655=1039.239,310.353,-118.596,171.877,42.737,158.225
C09656=1039.232,310.105,-118.562,171.873,42.735,158.225
C09657=1039.225,309.857,-118.529,171.869,42.733,158.224
C09658=1039.218,309.610,-118.495,171.865,42.731,158.223
C09659=1039.211,309.363,-118.461,171.861,42.728,158.222
C09660=1039.203,309.115,-118.428,171.857,42.727,158.222
C09661=1039.196,308.867,-118.395,171.853,42.725,158.221
C09662=1039.190,308.620,-118.362,171.848,42.723,158.220
C09663=1039.183,308.373,-118.328,171.844,42.721,158.220
C09664=1039.176,308.124,-118.295,171.840,42.719,158.219
C09665=1039.168,307.877,-118.261,171.836,42.717,158.218
C09666=1039.161,307.630,-118.228,171.832,42.715,158.217
C09667=1039.154,307.382,-118.194,171.828,42.713,158.217
C09668=1039.147,307.134,-118.161,171.824,42.712,158.216
C09669=1039.140,306.887,-118.128,171.820,42.710,158.215
C09670=1039.134,306.639,-118.094,171.815,42.708,158.214
C09671=1039.126,306.391,-118.061,171.811,42.706,158.214
C09672=1039.116,306.040,-118.014,171.806,42.703,158.213
C09673=1039.106,305.688,-117.967,171.800,42.701,158.212
C09674=1039.097,305.336,-117.920,171.795,42.698,158.211
C09675=1039.087,304.985,-117.872,171.788,42.695,158.210
C09676=1039.080,304.737,-117.839,171.784,42.693,158.209
C09677=1039.072,304.490,-117.806,171.781,42.691,158.208
C09678=1039.065,304.241,-117.773,171.776,42.689,158.207
C09679=1039.059,303.995,-117.739,171.772,42.688,158.207
C09680=1039.052,303.746,-117.706,171.768,42.686,158.206
C09681=1039.046,303.499,-117.673,171.764,42.684,158.205
C09682=1039.038,303.251,-117.639,171.761,42.682,158.205
C09683=1039.031,303.004,-117.607,171.757,42.680,158.204
C09684=1039.024,302.756,-117.574,171.753,42.678,158.203
C09685=1039.018,302.508,-117.541,171.748,42.677,158.203
C09686=1039.011,302.260,-117.508,171.744,42.675,158.202
C09687=1039.004,302.013,-117.475,171.740,42.673,158.201
C09688=1038.997,301.765,-117.442,171.736,42.671,158.200
C09689=1038.990,301.518,-117.409,171.733,42.669,158.200
C09690=1038.984,301.269,-117.376,171.729,42.668,158.199
C09691=1038.977,301.022,-117.342,171.725,42.666,158.198
C09692=1038.969,300.774,-117.310,171.721,42.664,158.198
C09693=1038.963,300.527,-117.277,171.717,42.662,158.197
C09694=1038.956,300.278,-117.244,171.713,42.660,158.196
C09695=1038.950,300.031,-117.211,171.709,42.658,158.196
C09696=1038.943,299.784,-117.178,171.705,42.657,158.195
C09697=1038.936,299.536,-117.145,171.701,42.655,158.194
C09698=1038.929,299.288,-117.113,171.697,42.653,158.194
C09699=1038.922,299.040,-117.079,171.693,42.651,158.193
C09700=1038.916,298.793,-117.046,171.690,42.649,158.192
C09701=1038.909,298.546,-117.014,171.686,42.648,158.192
C09702=1038.902,298.297,-116.981,171.682,42.646,158.191
C09703=1038.896,298.050,-116.948,171.678,42.644,158.190
C09704=1038.889,297.802,-116.915,171.674,42.642,158.190
C09705=1038.882,297.554,-116.883,171.671,42.640,158.189
C09706=1038.875,297.307,-116.850,171.667,42.639,158.188
C09707=1038.869,297.059,-116.817,171.663,42.637,158.188
C09708=1038.862,296.811,-116.784,171.659,42.635,158.187
C09709=1038.855,296.563,-116.752,171.655,42.633,158.186
C09710=1038.849,296.316,-116.719,171.652,42.631,158.186
C09711=1038.842,296.068,-116.686,171.648,42.629,158.185
C09712=1038.836,295.820,-116.653,171.644,42.627,158.184
C09713=1038.829,295.573,-116.621,171.640,42.626,158.184
C09714=1038.822,295.325,-116.588,171.637,42.624,158.183
C09715=1038.816,295.077,-116.555,171.633,42.622,158.182
C09716=1038.808,294.830,-116.523,171.629,42.621,158.182
C09717=1038.802,294.581,-116.491,171.625,42.619,158.181
C09718=1038.795,294.333,-116.459,171.621,42.617,158.180
C09719=1038.788,294.086,-116.427,171.617,42.616,158.180
C09720=1038.782,293.838,-116.394,171.613,42.614,158.179
C09721=1038.774,293.590,-116.362,171.609,42.613,158.178
C09722=1038.768,293.342,-116.329,171.605,42.611,158.178
C09723=1038.761,293.095,-116.297,171.602,42.609,158.177
C09724=1038.753,292.847,-116.265,171.598,42.607,158.176
C09725=1038.747,292.599,-116.233,171.594,42.606,158.176
C09726=1038.740,292.352,-116.200,171.590,42.604,158.175
C09727=1038.734,292.104,-116.169,171.587,42.603,158.175
C09728=1038.724,291.769,-116.125,171.582,42.600,158.174
C09729=1038.715,291.434,-116.081,171.577,42.598,158.173
C09730=1038.706,291.099,-116.038,171.572,42.596,158.172
C09731=1038.697,290.763,-115.994,171.567,42.594,158.171
C09732=1038.690,290.516,-115.962,171.563,42.592,158.171
C09733=1038.683,290.268,-115.931,171.559,42.590,158.170
C09734=1038.676,290.021,-115.899,171.556,42.589,158.169
C09735=1038.670,289.772,-115.866,171.553,42.587,158.169
C09736=1038.663,289.525,-115.834,171.549,42.586,158.168
C09737=1038.656,289.277,-115.803,171.546,42.584,158.168
C09738=1038.649,289.029,-115.770,171.542,42.582,158.167
C09739=1038.643,288.781,-115.739,171.538,42.581,158.166
C09740=1038.635,288.533,-115.707,171.534,42.580,158.166
C09741=1038.628,288.285,-115.675,171.531,42.578,158.165
C09742=1038.622,288.037,-115.643,171.527,42.576,158.164
C09743=1038.616,287.789,-115.611,171.523,42.574,158.164
C09744=1038.609,287.542,-115.579,171.519,42.573,158.163
C09745=1038.602,287.294,-115.548,171.516,42.572,158.163
C09746=1038.595,287.046,-115.516,171.512,42.570,158.162
C09747=1038.588,286.799,-115.484,171.508,42.568,158.161
C09748=1038.581,286.550,-115.452,171.505,42.567,158.161
C09749=1038.574,286.302,-115.421,171.502,42.566,158.160
C09750=1038.567,286.054,-115.389,171.498,42.564,158.160
C09751=1038.560,285.807,-115.357,171.495,42.562,158.159
C09752=1038.554,285.559,-115.326,171.491,42.561,158.158
C09753=1038.547,285.311,-115.294,171.487,42.560,158.158
C09754=1038.540,285.063,-115.263,171.484,42.558,158.157
C09755=1038.533,284.815,-115.231,171.480,42.556,158.157
C09756=1038.526,284.567,-115.200,171.476,42.555,158.156
C09757=1038.519,284.319,-115.168,171.473,42.554,158.156
C09758=1038.512,284.072,-115.136,171.469,42.552,158.155
C09759=1038.506,283.824,-115.105,171.466,42.550,158.154
C09760=1038.499,283.576,-115.073,171.463,42.549,158.154
C09761=1038.492,283.328,-115.042,171.459,42.547,158.153
C09762=1038.485,283.080,-115.010,171.455,42.546,158.153
C09763=1038.479,282.832,-114.979,171.452,42.545,158.152
C09764=1038.472,282.584,-114.948,171.448,42.543,158.152
C09765=1038.465,282.336,-114.916,171.444,42.541,158.151
C09766=1038.459,282.088,-114.885,171.442,42.540,158.150
C09767=1038.452,281.841,-114.853,171.438,42.538,158.150
C09768=1038.445,281.593,-114.822,171.434,42.537,158.149
C09769=1038.438,281.345,-114.790,171.431,42.536,158.149
C09770=1038.432,281.097,-114.759,171.427,42.534,158.148
C09771=1038.425,280.849,-114.727,171.423,42.532,158.147
C09772=1038.418,280.601,-114.696,171.421,42.531,158.147
C09773=1038.412,280.352,-114.665,171.417,42.530,158.146
C09774=1038.405,280.105,-114.634,171.413,42.528,158.146
C09775=1038.398,279.857,-114.602,171.410,42.527,158.145
C09776=1038.392,279.609,-114.571,171.406,42.525,158.145
C09777=1038.385,279.361,-114.540,171.402,42.524,158.144
C09778=1038.378,279.113,-114.508,171.400,42.523,158.144
C09779=1038.372,278.866,-114.477,171.396,42.521,158.143
C09780=1038.366,278.617,-114.446,171.392,42.519,158.142
C09781=1038.359,278.369,-114.415,171.389,42.518,158.142
C09782=1038.352,278.121,-114.384,171.386,42.516,158.141
C09783=1038.345,277.874,-114.353,171.382,42.515,158.141
C09784=1038.337,277.550,-114.313,171.378,42.513,158.140
C09785=1038.327,277.227,-114.272,171.373,42.511,158.139
C09786=1038.319,276.904,-114.232,171.369,42.510,158.139
C09787=1038.310,276.581,-114.192,171.364,42.508,158.138
C09788=1038.303,276.333,-114.160,171.361,42.507,158.137
C09789=1038.297,276.085,-114.129,171.358,42.505,158.137
C09790=1038.290,275.837,-114.098,171.354,42.504,158.136
C09791=1038.283,275.589,-114.068,171.351,42.503,158.136
C09792=1038.276,275.341,-114.036,171.347,42.501,158.135
C09793=1038.269,275.093,-114.005,171.344,42.500,158.135
C09794=1038.262,274.845,-113.975,171.341,42.498,158.134
C09795=1038.256,274.598,-113.944,171.337,42.497,158.134
C09796=1038.250,274.349,-113.913,171.334,42.496,158.133
C09797=1038.243,274.101,-113.882,171.331,42.494,158.133
C09798=1038.236,273.853,-113.852,171.327,42.493,158.132
C09799=1038.229,273.605,-113.820,171.324,42.491,158.131
C09800=1038.222,273.358,-113.790,171.320,42.490,158.131
C09801=1038.216,273.109,-113.760,171.317,42.489,158.130
C09802=1038.209,272.861,-113.728,171.314,42.487,158.130
C09803=1038.202,272.613,-113.698,171.310,42.486,158.129
C09804=1038.195,272.365,-113.667,171.307,42.485,158.129
C09805=1038.190,272.117,-113.636,171.304,42.484,158.128
C09806=1038.182,271.869,-113.606,171.300,42.482,158.128
C09807=1038.176,271.621,-113.575,171.297,42.481,158.127
C09808=1038.168,271.373,-113.545,171.294,42.479,158.127
C09809=1038.162,271.124,-113.514,171.291,42.478,158.126
C09810=1038.156,270.877,-113.483,171.287,42.477,158.126
C09811=1038.149,270.629,-113.453,171.283,42.476,158.125
C09812=1038.142,270.380,-113.422,171.281,42.474,158.125
C09813=1038.135,270.133,-113.391,171.277,42.473,158.124
C09814=1038.128,269.885,-113.361,171.274,42.472,158.124
C09815=1038.122,269.637,-113.331,171.271,42.470,158.123
C09816=1038.115,269.389,-113.301,171.268,42.469,158.123
C09817=1038.108,269.140,-113.270,171.264,42.468,158.122
C09818=1038.101,268.893,-113.239,171.261,42.466,158.122
C09819=1038.095,268.645,-113.209,171.258,42.465,158.121
C09820=1038.088,268.396,-113.179,171.254,42.464,158.121
C09821=1038.082,268.149,-113.148,171.252,42.463,158.120
C09822=1038.075,267.900,-113.118,171.248,42.461,158.120
C09823=1038.069,267.652,-113.087,171.244,42.460,158.119
C09824=1038.062,267.404,-113.058,171.242,42.458,158.119
C09825=1038.054,267.157,-113.027,171.238,42.458,158.118
C09826=1038.048,266.908,-112.996,171.235,42.456,158.118
C09827=1038.041,266.660,-112.966,171.232,42.455,158.117
C09828=1038.034,266.412,-112.936,171.228,42.453,158.117
C09829=1038.028,266.164,-112.905,171.225,42.453,158.116
C09830=1038.021,265.916,-112.875,171.222,42.451,158.116
C09831=1038.014,265.668,-112.846,171.219,42.450,158.115
C09832=1038.008,265.420,-112.815,171.215,42.449,158.115
C09833=1038.001,265.172,-112.785,171.213,42.447,158.114
C09834=1037.994,264.923,-112.756,171.209,42.446,158.114
C09835=1037.988,264.675,-112.725,171.206,42.445,158.113
C09836=1037.981,264.427,-112.695,171.203,42.444,158.113
C09837=1037.974,264.179,-112.665,171.199,42.442,158.112
C09838=1037.967,263.931,-112.635,171.197,42.441,158.112
C09839=1037.961,263.683,-112.605,171.193,42.440,158.111
C09840=1037.953,263.364,-112.566,171.190,42.438,158.111
C09841=1037.944,263.046,-112.528,171.185,42.437,158.110
C09842=1037.935,262.728,-112.489,171.181,42.435,158.109
C09843=1037.927,262.409,-112.450,171.177,42.434,158.109
C09844=1037.920,262.160,-112.420,171.174,42.432,158.108
C09845=1037.914,261.913,-112.391,171.171,42.431,158.108
C09846=1037.906,261.665,-112.360,171.168,42.430,158.107
C09847=1037.900,261.417,-112.331,171.164,42.429,158.107
C09848=1037.893,261.168,-112.301,171.162,42.428,158.106
C09849=1037.886,260.920,-112.271,171.158,42.427,158.106
C09850=1037.880,260.672,-112.242,171.155,42.425,158.105
C09851=1037.873,260.424,-112.212,171.152,42.425,158.105
C09852=1037.865,260.176,-112.182,171.149,42.423,158.104
C09853=1037.859,259.927,-112.153,171.146,42.422,158.104
C09854=1037.852,259.679,-112.123,171.143,42.421,158.104
C09855=1037.846,259.431,-112.094,171.139,42.420,158.103
C09856=1037.838,259.183,-112.064,171.137,42.419,158.103
C09857=1037.831,258.936,-112.034,171.133,42.418,158.102
C09858=1037.824,258.687,-112.005,171.131,42.416,158.102
C09859=1037.817,258.439,-111.975,171.127,42.415,158.101
C09860=1037.811,258.190,-111.946,171.123,42.414,158.101
C09861=1037.804,257.942,-111.916,171.121,42.413,158.100
C09862=1037.798,257.694,-111.887,171.117,42.412,158.100
C09863=1037.790,257.446,-111.857,171.115,42.411,158.100
C09864=1037.784,257.198,-111.828,171.111,42.410,158.099
C09865=1037.777,256.950,-111.797,171.109,42.409,158.099
C09866=1037.770,256.702,-111.769,171.106,42.408,158.098
C09867=1037.763,256.453,-111.740,171.103,42.406,158.098
C09868=1037.757,256.205,-111.710,171.099,42.406,158.097
C09869=1037.750,255.957,-111.680,171.096,42.404,158.097
C09870=1037.743,255.709,-111.651,171.093,42.403,158.096
C09871=1037.736,255.460,-111.621,171.090,42.402,158.096
C09872=1037.730,255.213,-111.591,171.087,42.401,158.095
C09873=1037.723,254.964,-111.562,171.084,42.400,158.095
C09874=1037.717,254.716,-111.533,171.081,42.399,158.095
C09875=1037.709,254.468,-111.504,171.078,42.397,158.094
C09876=1037.703,254.220,-111.474,171.075,42.396,158.094
C09877=1037.696,253.972,-111.445,171.072,42.396,158.093
C09878=1037.689,253.723,-111.415,171.069,42.394,158.093
C09879=1037.683,253.475,-111.386,171.066,42.393,158.092
C09880=1037.676,253.226,-111.357,171.063,42.392,158.092
C09881=1037.670,252.978,-111.328,171.060,42.391,158.091
C09882=1037.663,252.731,-111.298,171.057,42.389,158.091
C09883=1037.656,252.482,-111.269,171.054,42.389,158.091
C09884=1037.649,252.234,-111.240,171.051,42.387,158.090
C09885=1037.642,251.986,-111.210,171.048,42.386,158.090
C09886=1037.636,251.738,-111.181,171.045,42.385,158.089
C09887=1037.630,251.490,-111.152,171.042,42.384,158.089
C09888=1037.623,251.241,-111.123,171.039,42.383,158.088
C09889=1037.617,250.993,-111.094,171.037,42.381,158.088
C09890=1037.609,250.745,-111.064,171.033,42.381,158.087
C09891=1037.603,250.497,-111.035,171.031,42.379,158.087
C09892=1037.596,250.249,-111.006,171.027,42.378,158.087
C09893=1037.590,250.000,-110.977,171.025,42.377,158.086
C09894=1037.583,249.752,-110.948,171.021,42.376,158.086
C09895=1037.577,249.503,-110.918,171.019,42.375,158.085
C09896=1037.568,249.183,-110.881,171.015,42.374,158.085
C09897=1037.560,248.864,-110.843,171.011,42.372,158.084
C09898=1037.551,248.543,-110.806,171.008,42.370,158.083
C09899=1037.543,248.224,-110.768,171.003,42.369,158.083
C09900=1037.537,247.976,-110.739,171.001,42.368,158.083
C09901=1037.530,247.727,-110.710,170.998,42.367,158.082
C09902=1037.524,247.479,-110.681,170.995,42.366,158.082
C09903=1037.517,247.231,-110.653,170.992,42.365,158.081
C09904=1037.510,246.983,-110.623,170.989,42.364,158.081
C09905=1037.503,246.734,-110.594,170.986,42.363,158.080
C09906=1037.497,246.486,-110.565,170.984,42.361,158.080
C09907=1037.491,246.238,-110.536,170.980,42.360,158.079
C09908=1037.485,245.990,-110.507,170.977,42.359,158.079
C09909=1037.477,245.741,-110.478,170.974,42.358,158.079
C09910=1037.471,245.493,-110.449,170.972,42.357,158.078
C09911=1037.465,245.245,-110.420,170.969,42.356,158.078
C09912=1037.458,244.997,-110.391,170.966,42.355,158.077
C09913=1037.452,244.749,-110.362,170.963,42.354,158.077
C09914=1037.445,244.500,-110.333,170.961,42.352,158.076
C09915=1037.438,244.252,-110.304,170.957,42.351,158.076
C09916=1037.431,244.004,-110.276,170.955,42.351,158.076
C09917=1037.425,243.755,-110.247,170.951,42.349,158.075
C09918=1037.418,243.508,-110.219,170.949,42.348,158.075
C09919=1037.411,243.259,-110.190,170.946,42.347,158.074
C09920=1037.405,243.011,-110.160,170.943,42.346,158.074
C09921=1037.398,242.763,-110.132,170.940,42.345,158.073
C09922=1037.392,242.514,-110.104,170.938,42.344,158.073
C09923=1037.385,242.266,-110.075,170.934,42.343,158.073
C09924=1037.378,242.017,-110.046,170.932,42.342,158.072
C09925=1037.372,241.769,-110.018,170.929,42.341,158.072
C09926=1037.366,241.521,-109.989,170.926,42.340,158.071
C09927=1037.359,241.273,-109.961,170.923,42.338,158.071
C09928=1037.352,241.025,-109.932,170.921,42.338,158.071
C09929=1037.346,240.776,-109.903,170.918,42.337,158.070
C09930=1037.339,240.528,-109.874,170.915,42.336,158.070
C09931=1037.332,240.279,-109.847,170.911,42.334,158.069
C09932=1037.326,240.031,-109.818,170.909,42.333,158.069
C09933=1037.319,239.783,-109.789,170.907,42.333,158.068
C09934=1037.312,239.535,-109.762,170.903,42.332,158.068
C09935=1037.306,239.287,-109.732,170.901,42.331,158.068
C09936=1037.299,239.038,-109.704,170.898,42.330,158.067
C09937=1037.292,238.790,-109.676,170.895,42.328,158.067
C09938=1037.285,238.541,-109.648,170.892,42.328,158.066
C09939=1037.279,238.293,-109.619,170.890,42.327,158.066
C09940=1037.272,238.045,-109.591,170.887,42.326,158.066
C09941=1037.265,237.797,-109.563,170.884,42.325,158.065
C09942=1037.259,237.548,-109.535,170.882,42.324,158.065
C09943=1037.252,237.300,-109.506,170.878,42.323,158.064
C09944=1037.245,237.051,-109.478,170.876,42.322,158.064
C09945=1037.238,236.803,-109.450,170.873,42.321,158.064
C09946=1037.232,236.555,-109.421,170.871,42.320,158.063
C09947=1037.225,236.306,-109.394,170.867,42.319,158.063
C09948=1037.218,236.058,-109.365,170.865,42.318,158.063
C09949=1037.212,235.810,-109.337,170.862,42.316,158.062
C09950=1037.205,235.562,-109.308,170.859,42.316,158.062
C09951=1037.199,235.313,-109.281,170.857,42.315,158.061
C09952=1037.189,234.988,-109.244,170.853,42.313,158.061
C09953=1037.181,234.661,-109.207,170.850,42.313,158.060
C09954=1037.172,234.336,-109.170,170.846,42.311,158.060
C09955=1037.163,234.010,-109.133,170.842,42.310,158.059
C09956=1037.157,233.762,-109.105,170.840,42.309,158.059
C09957=1037.150,233.513,-109.077,170.837,42.308,158.059
C09958=1037.143,233.265,-109.048,170.834,42.306,158.058
C09959=1037.137,233.017,-109.021,170.831,42.306,158.058
C09960=1037.131,232.768,-108.992,170.829,42.305,158.057
C09961=1037.124,232.520,-108.965,170.827,42.304,158.057
C09962=1037.117,232.272,-108.936,170.823,42.303,158.057
C09963=1037.110,232.023,-108.908,170.821,42.302,158.056
C09964=1037.104,231.775,-108.881,170.818,42.301,158.056
C09965=1037.098,231.526,-108.852,170.816,42.299,158.055
C09966=1037.091,231.278,-108.824,170.812,42.299,158.055
C09967=1037.084,231.030,-108.796,170.810,42.298,158.055
C09968=1037.077,230.781,-108.768,170.808,42.297,158.054
C09969=1037.071,230.533,-108.741,170.805,42.296,158.054
C09970=1037.064,230.285,-108.713,170.802,42.295,158.053
C09971=1037.057,230.036,-108.685,170.799,42.294,158.053
C09972=1037.051,229.788,-108.658,170.797,42.293,158.053
C09973=1037.044,229.540,-108.629,170.794,42.292,158.052
C09974=1037.037,229.291,-108.601,170.791,42.291,158.052
C09975=1037.030,229.043,-108.574,170.788,42.290,158.051
C09976=1037.024,228.795,-108.546,170.786,42.289,158.051
C09977=1037.018,228.546,-108.518,170.784,42.288,158.051
C09978=1037.011,228.297,-108.490,170.781,42.287,158.050
C09979=1037.004,228.049,-108.462,170.778,42.286,158.050
C09980=1036.997,227.801,-108.435,170.775,42.285,158.050
C09981=1036.990,227.552,-108.407,170.773,42.284,158.049
C09982=1036.984,227.305,-108.380,170.771,42.283,158.049
C09983=1036.978,227.056,-108.352,170.768,42.283,158.049
C09984=1036.971,226.808,-108.324,170.765,42.282,158.048
C09985=1036.964,226.559,-108.297,170.762,42.281,158.048
C09986=1036.957,226.311,-108.269,170.760,42.280,158.047
C09987=1036.950,226.062,-108.243,170.757,42.279,158.047
C09988=1036.944,225.814,-108.215,170.754,42.278,158.047
C09989=1036.937,225.565,-108.187,170.752,42.277,158.046
C09990=1036.930,225.317,-108.159,170.749,42.276,158.046
C09991=1036.924,225.068,-108.132,170.747,42.275,158.046
C09992=1036.917,224.820,-108.104,170.744,42.274,158.045
C09993=1036.910,224.572,-108.077,170.742,42.273,158.045
C09994=1036.903,224.323,-108.050,170.739,42.273,158.044
C09995=1036.897,224.075,-108.022,170.736,42.272,158.044
C09996=1036.890,223.827,-107.995,170.734,42.271,158.044
//INST
///DATE 2021/06/17 10:58
///ATTR SC,RW,RJ
////FRAME ROBOT
///GROUP1 RB1
NOP
MOVL C00000 V=800.0 PL=0
MOVL C00001 V=800.0 PL=0
MOVL C00002 V=800.0 PL=0
MOVL C00003 V=800.0 PL=0
MOVL C00004 V=800.0 PL=0
MOVL C00005 V=800.0 PL=0
MOVL C00006 V=800.0 PL=0
MOVL C00007 V=800.0 PL=0
MOVL C00008 V=800.0 PL=0
MOVL C00009 V=800.0 PL=0
MOVL C00010 V=800.0 PL=0
MOVL C00011 V=800.0 PL=0
MOVL C00012 V=800.0 PL=0
MOVL C00013 V=800.0 PL=0
MOVL C00014 V=800.0 PL=0
MOVL C00015 V=800.0 PL=0
MOVL C00016 V=800.0 PL=0
MOVL C00017 V=800.0 PL=0
MOVL C00018 V=800.0 PL=0
MOVL C00019 V=800.0 PL=0
MOVL C00020 V=800.0 PL=0
MOVL C00021 V=800.0 PL=0
MOVL C00022 V=800.0 PL=0
MOVL C00023 V=800.0 PL=0
MOVL C00024 V=800.0 PL=0
MOVL C00025 V=800.0 PL=0
MOVL C00026 V=800.0 PL=0
MOVL C00027 V=800.0 PL=0
MOVL C00028 V=800.0 PL=0
MOVL C00029 V=800.0 PL=0
MOVL C00030 V=800.0 PL=0
MOVL C00031 V=800.0 PL=0
MOVL C00032 V=800.0 PL=0
MOVL C00033 V=800.0 PL=0
MOVL C00034 V=800.0 PL=0
MOVL C00035 V=800.0 PL=0
MOVL C00036 V=800.0 PL=0
MOVL C00037 V=800.0 PL=0
MOVL C00038 V=800.0 PL=0
MOVL C00039 V=800.0 PL=0
MOVL C00040 V=800.0 PL=0
MOVL C00041 V=800.0 PL=0
MOVL C00042 V=800.0 PL=0
MOVL C00043 V=800.0 PL=0
MOVL C00044 V=800.0 PL=0
MOVL C00045 V=800.0 PL=0
MOVL C00046 V=800.0 PL=0
MOVL C00047 V=800.0 PL=0
MOVL C00048 V=800.0 PL=0
MOVL C00049 V=800.0 PL=0
MOVL C00050 V=800.0 PL=0
MOVL C00051 V=800.0 PL=0
MOVL C00052 V=800.0 PL=0
MOVL C00053 V=800.0 PL=0
MOVL C00054 V=800.0 PL=0
MOVL C00055 V=800.0 PL=0
MOVL C00056 V=800.0 PL=0
MOVL C00057 V=800.0 PL=0
MOVL C00058 V=800.0 PL=0
MOVL C00059 V=800.0 PL=0
MOVL C00060 V=800.0 PL=0
MOVL C00061 V=800.0 PL=0
MOVL C00062 V=800.0 PL=0
MOVL C00063 V=800.0 PL=0
MOVL C00064 V=800.0 PL=0
MOVL C00065 V=800.0 PL=0
MOVL C00066 V=800.0 PL=0
MOVL C00067 V=800.0 PL=0
MOVL C00068 V=800.0 PL=0
MOVL C00069 V=800.0 PL=0
MOVL C00070 V=800.0 PL=0
MOVL C00071 V=800.0 PL=0
MOVL C00072 V=800.0 PL=0
MOVL C00073 V=800.0 PL=0
MOVL C00074 V=800.0 PL=0
MOVL C00075 V=800.0 PL=0
MOVL C00076 V=800.0 PL=0
MOVL C00077 V=800.0 PL=0
MOVL C00078 V=800.0 PL=0
MOVL C00079 V=800.0 PL=0
MOVL C00080 V=800.0 PL=0
MOVL C00081 V=800.0 PL=0
MOVL C00082 V=800.0 PL=0
MOVL C00083 V=800.0 PL=0
MOVL C00084 V=800.0 PL=0
MOVL C00085 V=800.0 PL=0
MOVL C00086 V=800.0 PL=0
MOVL C00087 V=800.0 PL=0
MOVL C00088 V=800.0 PL=0
MOVL C00089 V=800.0 PL=0
MOVL C00090 V=800.0 PL=0
MOVL C00091 V=800.0 PL=0
MOVL C00092 V=800.0 PL=0
MOVL C00093 V=800.0 PL=0
MOVL C00094 V=800.0 PL=0
MOVL C00095 V=800.0 PL=0
MOVL C00096 V=800.0 PL=0
MOVL C00097 V=800.0 PL=0
MOVL C00098 V=800.0 PL=0
MOVL C00099 V=800.0 PL=0
MOVL C00100 V=800.0 PL=0
MOVL C00101 V=800.0 PL=0
MOVL C00102 V=800.0 PL=0
MOVL C00103 V=800.0 PL=0
MOVL C00104 V=800.0 PL=0
MOVL C00105 V=800.0 PL=0
MOVL C00106 V=800.0 PL=0
MOVL C00107 V=800.0 PL=0
MOVL C00108 V=800.0 PL=0
MOVL C00109 V=800.0 PL=0
MOVL C00110 V=800.0 PL=0
MOVL C00111 V=800.0 PL=0
MOVL C00112 V=800.0 PL=0
MOVL C00113 V=800.0 PL=0
MOVL C00114 V=800.0 PL=0
MOVL C00115 V=800.0 PL=0
MOVL C00116 V=800.0 PL=0
MOVL C00117 V=800.0 PL=0
MOVL C00118 V=800.0 PL=0
MOVL C00119 V=800.0 PL=0
MOVL C00120 V=800.0 PL=0
MOVL C00121 V=800.0 PL=0
MOVL C00122 V=800.0 PL=0
MOVL C00123 V=800.0 PL=0
MOVL C00124 V=800.0 PL=0
MOVL C00125 V=800.0 PL=0
MOVL C00126 V=800.0 PL=0
MOVL C00127 V=800.0 PL=0
MOVL C00128 V=800.0 PL=0
MOVL C00129 V=800.0 PL=0
MOVL C00130 V=800.0 PL=0
MOVL C00131 V=800.0 PL=0
MOVL C00132 V=800.0 PL=0
MOVL C00133 V=800.0 PL=0
MOVL C00134 V=800.0 PL=0
MOVL C00135 V=800.0 PL=0
MOVL C00136 V=800.0 PL=0
MOVL C00137 V=800.0 PL=0
MOVL C00138 V=800.0 PL=0
MOVL C00139 V=800.0 PL=0
MOVL C00140 V=800.0 PL=0
MOVL C00141 V=800.0 PL=0
MOVL C00142 V=800.0 PL=0
MOVL C00143 V=800.0 PL=0
MOVL C00144 V=800.0 PL=0
MOVL C00145 V=800.0 PL=0
MOVL C00146 V=800.0 PL=0
MOVL C00147 V=800.0 PL=0
MOVL C00148 V=800.0 PL=0
MOVL C00149 V=800.0 PL=0
MOVL C00150 V=800.0 PL=0
MOVL C00151 V=800.0 PL=0
MOVL C00152 V=800.0 PL=0
MOVL C00153 V=800.0 PL=0
MOVL C00154 V=800.0 PL=0
MOVL C00155 V=800.0 PL=0
MOVL C00156 V=800.0 PL=0
MOVL C00157 V=800.0 PL=0
MOVL C00158 V=800.0 PL=0
MOVL C00159 V=800.0 PL=0
MOVL C00160 V=800.0 PL=0
MOVL C00161 V=800.0 PL=0
MOVL C00162 V=800.0 PL=0
MOVL C00163 V=800.0 PL=0
MOVL C00164 V=800.0 PL=0
MOVL C00165 V=800.0 PL=0
MOVL C00166 V=800.0 PL=0
MOVL C00167 V=800.0 PL=0
MOVL C00168 V=800.0 PL=0
MOVL C00169 V=800.0 PL=0
MOVL C00170 V=800.0 PL=0
MOVL C00171 V=800.0 PL=0
MOVL C00172 V=800.0 PL=0
MOVL C00173 V=800.0 PL=0
MOVL C00174 V=800.0 PL=0
MOVL C00175 V=800.0 PL=0
MOVL C00176 V=800.0 PL=0
MOVL C00177 V=800.0 PL=0
MOVL C00178 V=800.0 PL=0
MOVL C00179 V=800.0 PL=0
MOVL C00180 V=800.0 PL=0
MOVL C00181 V=800.0 PL=0
MOVL C00182 V=800.0 PL=0
MOVL C00183 V=800.0 PL=0
MOVL C00184 V=800.0 PL=0
MOVL C00185 V=800.0 PL=0
MOVL C00186 V=800.0 PL=0
MOVL C00187 V=800.0 PL=0
MOVL C00188 V=800.0 PL=0
MOVL C00189 V=800.0 PL=0
MOVL C00190 V=800.0 PL=0
MOVL C00191 V=800.0 PL=0
MOVL C00192 V=800.0 PL=0
MOVL C00193 V=800.0 PL=0
MOVL C00194 V=800.0 PL=0
MOVL C00195 V=800.0 PL=0
MOVL C00196 V=800.0 PL=0
MOVL C00197 V=800.0 PL=0
MOVL C00198 V=800.0 PL=0
MOVL C00199 V=800.0 PL=0
MOVL C00200 V=800.0 PL=0
MOVL C00201 V=800.0 PL=0
MOVL C00202 V=800.0 PL=0
MOVL C00203 V=800.0 PL=0
MOVL C00204 V=800.0 PL=0
MOVL C00205 V=800.0 PL=0
MOVL C00206 V=800.0 PL=0
MOVL C00207 V=800.0 PL=0
MOVL C00208 V=800.0 PL=0
MOVL C00209 V=800.0 PL=0
MOVL C00210 V=800.0 PL=0
MOVL C00211 V=800.0 PL=0
MOVL C00212 V=800.0 PL=0
MOVL C00213 V=800.0 PL=0
MOVL C00214 V=800.0 PL=0
MOVL C00215 V=800.0 PL=0
MOVL C00216 V=800.0 PL=0
MOVL C00217 V=800.0 PL=0
MOVL C00218 V=800.0 PL=0
MOVL C00219 V=800.0 PL=0
MOVL C00220 V=800.0 PL=0
MOVL C00221 V=800.0 PL=0
MOVL C00222 V=800.0 PL=0
MOVL C00223 V=800.0 PL=0
MOVL C00224 V=800.0 PL=0
MOVL C00225 V=800.0 PL=0
MOVL C00226 V=800.0 PL=0
MOVL C00227 V=800.0 PL=0
MOVL C00228 V=800.0 PL=0
MOVL C00229 V=800.0 PL=0
MOVL C00230 V=800.0 PL=0
MOVL C00231 V=800.0 PL=0
MOVL C00232 V=800.0 PL=0
MOVL C00233 V=800.0 PL=0
MOVL C00234 V=800.0 PL=0
MOVL C00235 V=800.0 PL=0
MOVL C00236 V=800.0 PL=0
MOVL C00237 V=800.0 PL=0
MOVL C00238 V=800.0 PL=0
MOVL C00239 V=800.0 PL=0
MOVL C00240 V=800.0 PL=0
MOVL C00241 V=800.0 PL=0
MOVL C00242 V=800.0 PL=0
MOVL C00243 V=800.0 PL=0
MOVL C00244 V=800.0 PL=0
MOVL C00245 V=800.0 PL=0
MOVL C00246 V=800.0 PL=0
MOVL C00247 V=800.0 PL=0
MOVL C00248 V=800.0 PL=0
MOVL C00249 V=800.0 PL=0
MOVL C00250 V=800.0 PL=0
MOVL C00251 V=800.0 PL=0
MOVL C00252 V=800.0 PL=0
MOVL C00253 V=800.0 PL=0
MOVL C00254 V=800.0 PL=0
MOVL C00255 V=800.0 PL=0
MOVL C00256 V=800.0 PL=0
MOVL C00257 V=800.0 PL=0
MOVL C00258 V=800.0 PL=0
MOVL C00259 V=800.0 PL=0
MOVL C00260 V=800.0 PL=0
MOVL C00261 V=800.0 PL=0
MOVL C00262 V=800.0 PL=0
MOVL C00263 V=800.0 PL=0
MOVL C00264 V=800.0 PL=0
MOVL C00265 V=800.0 PL=0
MOVL C00266 V=800.0 PL=0
MOVL C00267 V=800.0 PL=0
MOVL C00268 V=800.0 PL=0
MOVL C00269 V=800.0 PL=0
MOVL C00270 V=800.0 PL=0
MOVL C00271 V=800.0 PL=0
MOVL C00272 V=800.0 PL=0
MOVL C00273 V=800.0 PL=0
MOVL C00274 V=800.0 PL=0
MOVL C00275 V=800.0 PL=0
MOVL C00276 V=800.0 PL=0
MOVL C00277 V=800.0 PL=0
MOVL C00278 V=800.0 PL=0
MOVL C00279 V=800.0 PL=0
MOVL C00280 V=800.0 PL=0
MOVL C00281 V=800.0 PL=0
MOVL C00282 V=800.0 PL=0
MOVL C00283 V=800.0 PL=0
MOVL C00284 V=800.0 PL=0
MOVL C00285 V=800.0 PL=0
MOVL C00286 V=800.0 PL=0
MOVL C00287 V=800.0 PL=0
MOVL C00288 V=800.0 PL=0
MOVL C00289 V=800.0 PL=0
MOVL C00290 V=800.0 PL=0
MOVL C00291 V=800.0 PL=0
MOVL C00292 V=800.0 PL=0
MOVL C00293 V=800.0 PL=0
MOVL C00294 V=800.0 PL=0
MOVL C00295 V=800.0 PL=0
MOVL C00296 V=800.0 PL=0
MOVL C00297 V=800.0 PL=0
MOVL C00298 V=800.0 PL=0
MOVL C00299 V=800.0 PL=0
MOVL C00300 V=800.0 PL=0
MOVL C00301 V=800.0 PL=0
MOVL C00302 V=800.0 PL=0
MOVL C00303 V=800.0 PL=0
MOVL C00304 V=800.0 PL=0
MOVL C00305 V=800.0 PL=0
MOVL C00306 V=800.0 PL=0
MOVL C00307 V=800.0 PL=0
MOVL C00308 V=800.0 PL=0
MOVL C00309 V=800.0 PL=0
MOVL C00310 V=800.0 PL=0
MOVL C00311 V=800.0 PL=0
MOVL C00312 V=800.0 PL=0
MOVL C00313 V=800.0 PL=0
MOVL C00314 V=800.0 PL=0
MOVL C00315 V=800.0 PL=0
MOVL C00316 V=800.0 PL=0
MOVL C00317 V=800.0 PL=0
MOVL C00318 V=800.0 PL=0
MOVL C00319 V=800.0 PL=0
MOVL C00320 V=800.0 PL=0
MOVL C00321 V=800.0 PL=0
MOVL C00322 V=800.0 PL=0
MOVL C00323 V=800.0 PL=0
MOVL C00324 V=800.0 PL=0
MOVL C00325 V=800.0 PL=0
MOVL C00326 V=800.0 PL=0
MOVL C00327 V=800.0 PL=0
MOVL C00328 V=800.0 PL=0
MOVL C00329 V=800.0 PL=0
MOVL C00330 V=800.0 PL=0
MOVL C00331 V=800.0 PL=0
MOVL C00332 V=800.0 PL=0
MOVL C00333 V=800.0 PL=0
MOVL C00334 V=800.0 PL=0
MOVL C00335 V=800.0 PL=0
MOVL C00336 V=800.0 PL=0
MOVL C00337 V=800.0 PL=0
MOVL C00338 V=800.0 PL=0
MOVL C00339 V=800.0 PL=0
MOVL C00340 V=800.0 PL=0
MOVL C00341 V=800.0 PL=0
MOVL C00342 V=800.0 PL=0
MOVL C00343 V=800.0 PL=0
MOVL C00344 V=800.0 PL=0
MOVL C00345 V=800.0 PL=0
MOVL C00346 V=800.0 PL=0
MOVL C00347 V=800.0 PL=0
MOVL C00348 V=800.0 PL=0
MOVL C00349 V=800.0 PL=0
MOVL C00350 V=800.0 PL=0
MOVL C00351 V=800.0 PL=0
MOVL C00352 V=800.0 PL=0
MOVL C00353 V=800.0 PL=0
MOVL C00354 V=800.0 PL=0
MOVL C00355 V=800.0 PL=0
MOVL C00356 V=800.0 PL=0
MOVL C00357 V=800.0 PL=0
MOVL C00358 V=800.0 PL=0
MOVL C00359 V=800.0 PL=0
MOVL C00360 V=800.0 PL=0
MOVL C00361 V=800.0 PL=0
MOVL C00362 V=800.0 PL=0
MOVL C00363 V=800.0 PL=0
MOVL C00364 V=800.0 PL=0
MOVL C00365 V=800.0 PL=0
MOVL C00366 V=800.0 PL=0
MOVL C00367 V=800.0 PL=0
MOVL C00368 V=800.0 PL=0
MOVL C00369 V=800.0 PL=0
MOVL C00370 V=800.0 PL=0
MOVL C00371 V=800.0 PL=0
MOVL C00372 V=800.0 PL=0
MOVL C00373 V=800.0 PL=0
MOVL C00374 V=800.0 PL=0
MOVL C00375 V=800.0 PL=0
MOVL C00376 V=800.0 PL=0
MOVL C00377 V=800.0 PL=0
MOVL C00378 V=800.0 PL=0
MOVL C00379 V=800.0 PL=0
MOVL C00380 V=800.0 PL=0
MOVL C00381 V=800.0 PL=0
MOVL C00382 V=800.0 PL=0
MOVL C00383 V=800.0 PL=0
MOVL C00384 V=800.0 PL=0
MOVL C00385 V=800.0 PL=0
MOVL C00386 V=800.0 PL=0
MOVL C00387 V=800.0 PL=0
MOVL C00388 V=800.0 PL=0
MOVL C00389 V=800.0 PL=0
MOVL C00390 V=800.0 PL=0
MOVL C00391 V=800.0 PL=0
MOVL C00392 V=800.0 PL=0
MOVL C00393 V=800.0 PL=0
MOVL C00394 V=800.0 PL=0
MOVL C00395 V=800.0 PL=0
MOVL C00396 V=800.0 PL=0
MOVL C00397 V=800.0 PL=0
MOVL C00398 V=800.0 PL=0
MOVL C00399 V=800.0 PL=0
MOVL C00400 V=800.0 PL=0
MOVL C00401 V=800.0 PL=0
MOVL C00402 V=800.0 PL=0
MOVL C00403 V=800.0 PL=0
MOVL C00404 V=800.0 PL=0
MOVL C00405 V=800.0 PL=0
MOVL C00406 V=800.0 PL=0
MOVL C00407 V=800.0 PL=0
MOVL C00408 V=800.0 PL=0
MOVL C00409 V=800.0 PL=0
MOVL C00410 V=800.0 PL=0
MOVL C00411 V=800.0 PL=0
MOVL C00412 V=800.0 PL=0
MOVL C00413 V=800.0 PL=0
MOVL C00414 V=800.0 PL=0
MOVL C00415 V=800.0 PL=0
MOVL C00416 V=800.0 PL=0
MOVL C00417 V=800.0 PL=0
MOVL C00418 V=800.0 PL=0
MOVL C00419 V=800.0 PL=0
MOVL C00420 V=800.0 PL=0
MOVL C00421 V=800.0 PL=0
MOVL C00422 V=800.0 PL=0
MOVL C00423 V=800.0 PL=0
MOVL C00424 V=800.0 PL=0
MOVL C00425 V=800.0 PL=0
MOVL C00426 V=800.0 PL=0
MOVL C00427 V=800.0 PL=0
MOVL C00428 V=800.0 PL=0
MOVL C00429 V=800.0 PL=0
MOVL C00430 V=800.0 PL=0
MOVL C00431 V=800.0 PL=0
MOVL C00432 V=800.0 PL=0
MOVL C00433 V=800.0 PL=0
MOVL C00434 V=800.0 PL=0
MOVL C00435 V=800.0 PL=0
MOVL C00436 V=800.0 PL=0
MOVL C00437 V=800.0 PL=0
MOVL C00438 V=800.0 PL=0
MOVL C00439 V=800.0 PL=0
MOVL C00440 V=800.0 PL=0
MOVL C00441 V=800.0 PL=0
MOVL C00442 V=800.0 PL=0
MOVL C00443 V=800.0 PL=0
MOVL C00444 V=800.0 PL=0
MOVL C00445 V=800.0 PL=0
MOVL C00446 V=800.0 PL=0
MOVL C00447 V=800.0 PL=0
MOVL C00448 V=800.0 PL=0
MOVL C00449 V=800.0 PL=0
MOVL C00450 V=800.0 PL=0
MOVL C00451 V=800.0 PL=0
MOVL C00452 V=800.0 PL=0
MOVL C00453 V=800.0 PL=0
MOVL C00454 V=800.0 PL=0
MOVL C00455 V=800.0 PL=0
MOVL C00456 V=800.0 PL=0
MOVL C00457 V=800.0 PL=0
MOVL C00458 V=800.0 PL=0
MOVL C00459 V=800.0 PL=0
MOVL C00460 V=800.0 PL=0
MOVL C00461 V=800.0 PL=0
MOVL C00462 V=800.0 PL=0
MOVL C00463 V=800.0 PL=0
MOVL C00464 V=800.0 PL=0
MOVL C00465 V=800.0 PL=0
MOVL C00466 V=800.0 PL=0
MOVL C00467 V=800.0 PL=0
MOVL C00468 V=800.0 PL=0
MOVL C00469 V=800.0 PL=0
MOVL C00470 V=800.0 PL=0
MOVL C00471 V=800.0 PL=0
MOVL C00472 V=800.0 PL=0
MOVL C00473 V=800.0 PL=0
MOVL C00474 V=800.0 PL=0
MOVL C00475 V=800.0 PL=0
MOVL C00476 V=800.0 PL=0
MOVL C00477 V=800.0 PL=0
MOVL C00478 V=800.0 PL=0
MOVL C00479 V=800.0 PL=0
MOVL C00480 V=800.0 PL=0
MOVL C00481 V=800.0 PL=0
MOVL C00482 V=800.0 PL=0
MOVL C00483 V=800.0 PL=0
MOVL C00484 V=800.0 PL=0
MOVL C00485 V=800.0 PL=0
MOVL C00486 V=800.0 PL=0
MOVL C00487 V=800.0 PL=0
MOVL C00488 V=800.0 PL=0
MOVL C00489 V=800.0 PL=0
MOVL C00490 V=800.0 PL=0
MOVL C00491 V=800.0 PL=0
MOVL C00492 V=800.0 PL=0
MOVL C00493 V=800.0 PL=0
MOVL C00494 V=800.0 PL=0
MOVL C00495 V=800.0 PL=0
MOVL C00496 V=800.0 PL=0
MOVL C00497 V=800.0 PL=0
MOVL C00498 V=800.0 PL=0
MOVL C00499 V=800.0 PL=0
MOVL C00500 V=800.0 PL=0
MOVL C00501 V=800.0 PL=0
MOVL C00502 V=800.0 PL=0
MOVL C00503 V=800.0 PL=0
MOVL C00504 V=800.0 PL=0
MOVL C00505 V=800.0 PL=0
MOVL C00506 V=800.0 PL=0
MOVL C00507 V=800.0 PL=0
MOVL C00508 V=800.0 PL=0
MOVL C00509 V=800.0 PL=0
MOVL C00510 V=800.0 PL=0
MOVL C00511 V=800.0 PL=0
MOVL C00512 V=800.0 PL=0
MOVL C00513 V=800.0 PL=0
MOVL C00514 V=800.0 PL=0
MOVL C00515 V=800.0 PL=0
MOVL C00516 V=800.0 PL=0
MOVL C00517 V=800.0 PL=0
MOVL C00518 V=800.0 PL=0
MOVL C00519 V=800.0 PL=0
MOVL C00520 V=800.0 PL=0
MOVL C00521 V=800.0 PL=0
MOVL C00522 V=800.0 PL=0
MOVL C00523 V=800.0 PL=0
MOVL C00524 V=800.0 PL=0
MOVL C00525 V=800.0 PL=0
MOVL C00526 V=800.0 PL=0
MOVL C00527 V=800.0 PL=0
MOVL C00528 V=800.0 PL=0
MOVL C00529 V=800.0 PL=0
MOVL C00530 V=800.0 PL=0
MOVL C00531 V=800.0 PL=0
MOVL C00532 V=800.0 PL=0
MOVL C00533 V=800.0 PL=0
MOVL C00534 V=800.0 PL=0
MOVL C00535 V=800.0 PL=0
MOVL C00536 V=800.0 PL=0
MOVL C00537 V=800.0 PL=0
MOVL C00538 V=800.0 PL=0
MOVL C00539 V=800.0 PL=0
MOVL C00540 V=800.0 PL=0
MOVL C00541 V=800.0 PL=0
MOVL C00542 V=800.0 PL=0
MOVL C00543 V=800.0 PL=0
MOVL C00544 V=800.0 PL=0
MOVL C00545 V=800.0 PL=0
MOVL C00546 V=800.0 PL=0
MOVL C00547 V=800.0 PL=0
MOVL C00548 V=800.0 PL=0
MOVL C00549 V=800.0 PL=0
MOVL C00550 V=800.0 PL=0
MOVL C00551 V=800.0 PL=0
MOVL C00552 V=800.0 PL=0
MOVL C00553 V=800.0 PL=0
MOVL C00554 V=800.0 PL=0
MOVL C00555 V=800.0 PL=0
MOVL C00556 V=800.0 PL=0
MOVL C00557 V=800.0 PL=0
MOVL C00558 V=800.0 PL=0
MOVL C00559 V=800.0 PL=0
MOVL C00560 V=800.0 PL=0
MOVL C00561 V=800.0 PL=0
MOVL C00562 V=800.0 PL=0
MOVL C00563 V=800.0 PL=0
MOVL C00564 V=800.0 PL=0
MOVL C00565 V=800.0 PL=0
MOVL C00566 V=800.0 PL=0
MOVL C00567 V=800.0 PL=0
MOVL C00568 V=800.0 PL=0
MOVL C00569 V=800.0 PL=0
MOVL C00570 V=800.0 PL=0
MOVL C00571 V=800.0 PL=0
MOVL C00572 V=800.0 PL=0
MOVL C00573 V=800.0 PL=0
MOVL C00574 V=800.0 PL=0
MOVL C00575 V=800.0 PL=0
MOVL C00576 V=800.0 PL=0
MOVL C00577 V=800.0 PL=0
MOVL C00578 V=800.0 PL=0
MOVL C00579 V=800.0 PL=0
MOVL C00580 V=800.0 PL=0
MOVL C00581 V=800.0 PL=0
MOVL C00582 V=800.0 PL=0
MOVL C00583 V=800.0 PL=0
MOVL C00584 V=800.0 PL=0
MOVL C00585 V=800.0 PL=0
MOVL C00586 V=800.0 PL=0
MOVL C00587 V=800.0 PL=0
MOVL C00588 V=800.0 PL=0
MOVL C00589 V=800.0 PL=0
MOVL C00590 V=800.0 PL=0
MOVL C00591 V=800.0 PL=0
MOVL C00592 V=800.0 PL=0
MOVL C00593 V=800.0 PL=0
MOVL C00594 V=800.0 PL=0
MOVL C00595 V=800.0 PL=0
MOVL C00596 V=800.0 PL=0
MOVL C00597 V=800.0 PL=0
MOVL C00598 V=800.0 PL=0
MOVL C00599 V=800.0 PL=0
MOVL C00600 V=800.0 PL=0
MOVL C00601 V=800.0 PL=0
MOVL C00602 V=800.0 PL=0
MOVL C00603 V=800.0 PL=0
MOVL C00604 V=800.0 PL=0
MOVL C00605 V=800.0 PL=0
MOVL C00606 V=800.0 PL=0
MOVL C00607 V=800.0 PL=0
MOVL C00608 V=800.0 PL=0
MOVL C00609 V=800.0 PL=0
MOVL C00610 V=800.0 PL=0
MOVL C00611 V=800.0 PL=0
MOVL C00612 V=800.0 PL=0
MOVL C00613 V=800.0 PL=0
MOVL C00614 V=800.0 PL=0
MOVL C00615 V=800.0 PL=0
MOVL C00616 V=800.0 PL=0
MOVL C00617 V=800.0 PL=0
MOVL C00618 V=800.0 PL=0
MOVL C00619 V=800.0 PL=0
MOVL C00620 V=800.0 PL=0
MOVL C00621 V=800.0 PL=0
MOVL C00622 V=800.0 PL=0
MOVL C00623 V=800.0 PL=0
MOVL C00624 V=800.0 PL=0
MOVL C00625 V=800.0 PL=0
MOVL C00626 V=800.0 PL=0
MOVL C00627 V=800.0 PL=0
MOVL C00628 V=800.0 PL=0
MOVL C00629 V=800.0 PL=0
MOVL C00630 V=800.0 PL=0
MOVL C00631 V=800.0 PL=0
MOVL C00632 V=800.0 PL=0
MOVL C00633 V=800.0 PL=0
MOVL C00634 V=800.0 PL=0
MOVL C00635 V=800.0 PL=0
MOVL C00636 V=800.0 PL=0
MOVL C00637 V=800.0 PL=0
MOVL C00638 V=800.0 PL=0
MOVL C00639 V=800.0 PL=0
MOVL C00640 V=800.0 PL=0
MOVL C00641 V=800.0 PL=0
MOVL C00642 V=800.0 PL=0
MOVL C00643 V=800.0 PL=0
MOVL C00644 V=800.0 PL=0
MOVL C00645 V=800.0 PL=0
MOVL C00646 V=800.0 PL=0
MOVL C00647 V=800.0 PL=0
MOVL C00648 V=800.0 PL=0
MOVL C00649 V=800.0 PL=0
MOVL C00650 V=800.0 PL=0
MOVL C00651 V=800.0 PL=0
MOVL C00652 V=800.0 PL=0
MOVL C00653 V=800.0 PL=0
MOVL C00654 V=800.0 PL=0
MOVL C00655 V=800.0 PL=0
MOVL C00656 V=800.0 PL=0
MOVL C00657 V=800.0 PL=0
MOVL C00658 V=800.0 PL=0
MOVL C00659 V=800.0 PL=0
MOVL C00660 V=800.0 PL=0
MOVL C00661 V=800.0 PL=0
MOVL C00662 V=800.0 PL=0
MOVL C00663 V=800.0 PL=0
MOVL C00664 V=800.0 PL=0
MOVL C00665 V=800.0 PL=0
MOVL C00666 V=800.0 PL=0
MOVL C00667 V=800.0 PL=0
MOVL C00668 V=800.0 PL=0
MOVL C00669 V=800.0 PL=0
MOVL C00670 V=800.0 PL=0
MOVL C00671 V=800.0 PL=0
MOVL C00672 V=800.0 PL=0
MOVL C00673 V=800.0 PL=0
MOVL C00674 V=800.0 PL=0
MOVL C00675 V=800.0 PL=0
MOVL C00676 V=800.0 PL=0
MOVL C00677 V=800.0 PL=0
MOVL C00678 V=800.0 PL=0
MOVL C00679 V=800.0 PL=0
MOVL C00680 V=800.0 PL=0
MOVL C00681 V=800.0 PL=0
MOVL C00682 V=800.0 PL=0
MOVL C00683 V=800.0 PL=0
MOVL C00684 V=800.0 PL=0
MOVL C00685 V=800.0 PL=0
MOVL C00686 V=800.0 PL=0
MOVL C00687 V=800.0 PL=0
MOVL C00688 V=800.0 PL=0
MOVL C00689 V=800.0 PL=0
MOVL C00690 V=800.0 PL=0
MOVL C00691 V=800.0 PL=0
MOVL C00692 V=800.0 PL=0
MOVL C00693 V=800.0 PL=0
MOVL C00694 V=800.0 PL=0
MOVL C00695 V=800.0 PL=0
MOVL C00696 V=800.0 PL=0
MOVL C00697 V=800.0 PL=0
MOVL C00698 V=800.0 PL=0
MOVL C00699 V=800.0 PL=0
MOVL C00700 V=800.0 PL=0
MOVL C00701 V=800.0 PL=0
MOVL C00702 V=800.0 PL=0
MOVL C00703 V=800.0 PL=0
MOVL C00704 V=800.0 PL=0
MOVL C00705 V=800.0 PL=0
MOVL C00706 V=800.0 PL=0
MOVL C00707 V=800.0 PL=0
MOVL C00708 V=800.0 PL=0
MOVL C00709 V=800.0 PL=0
MOVL C00710 V=800.0 PL=0
MOVL C00711 V=800.0 PL=0
MOVL C00712 V=800.0 PL=0
MOVL C00713 V=800.0 PL=0
MOVL C00714 V=800.0 PL=0
MOVL C00715 V=800.0 PL=0
MOVL C00716 V=800.0 PL=0
MOVL C00717 V=800.0 PL=0
MOVL C00718 V=800.0 PL=0
MOVL C00719 V=800.0 PL=0
MOVL C00720 V=800.0 PL=0
MOVL C00721 V=800.0 PL=0
MOVL C00722 V=800.0 PL=0
MOVL C00723 V=800.0 PL=0
MOVL C00724 V=800.0 PL=0
MOVL C00725 V=800.0 PL=0
MOVL C00726 V=800.0 PL=0
MOVL C00727 V=800.0 PL=0
MOVL C00728 V=800.0 PL=0
MOVL C00729 V=800.0 PL=0
MOVL C00730 V=800.0 PL=0
MOVL C00731 V=800.0 PL=0
MOVL C00732 V=800.0 PL=0
MOVL C00733 V=800.0 PL=0
MOVL C00734 V=800.0 PL=0
MOVL C00735 V=800.0 PL=0
MOVL C00736 V=800.0 PL=0
MOVL C00737 V=800.0 PL=0
MOVL C00738 V=800.0 PL=0
MOVL C00739 V=800.0 PL=0
MOVL C00740 V=800.0 PL=0
MOVL C00741 V=800.0 PL=0
MOVL C00742 V=800.0 PL=0
MOVL C00743 V=800.0 PL=0
MOVL C00744 V=800.0 PL=0
MOVL C00745 V=800.0 PL=0
MOVL C00746 V=800.0 PL=0
MOVL C00747 V=800.0 PL=0
MOVL C00748 V=800.0 PL=0
MOVL C00749 V=800.0 PL=0
MOVL C00750 V=800.0 PL=0
MOVL C00751 V=800.0 PL=0
MOVL C00752 V=800.0 PL=0
MOVL C00753 V=800.0 PL=0
MOVL C00754 V=800.0 PL=0
MOVL C00755 V=800.0 PL=0
MOVL C00756 V=800.0 PL=0
MOVL C00757 V=800.0 PL=0
MOVL C00758 V=800.0 PL=0
MOVL C00759 V=800.0 PL=0
MOVL C00760 V=800.0 PL=0
MOVL C00761 V=800.0 PL=0
MOVL C00762 V=800.0 PL=0
MOVL C00763 V=800.0 PL=0
MOVL C00764 V=800.0 PL=0
MOVL C00765 V=800.0 PL=0
MOVL C00766 V=800.0 PL=0
MOVL C00767 V=800.0 PL=0
MOVL C00768 V=800.0 PL=0
MOVL C00769 V=800.0 PL=0
MOVL C00770 V=800.0 PL=0
MOVL C00771 V=800.0 PL=0
MOVL C00772 V=800.0 PL=0
MOVL C00773 V=800.0 PL=0
MOVL C00774 V=800.0 PL=0
MOVL C00775 V=800.0 PL=0
MOVL C00776 V=800.0 PL=0
MOVL C00777 V=800.0 PL=0
MOVL C00778 V=800.0 PL=0
MOVL C00779 V=800.0 PL=0
MOVL C00780 V=800.0 PL=0
MOVL C00781 V=800.0 PL=0
MOVL C00782 V=800.0 PL=0
MOVL C00783 V=800.0 PL=0
MOVL C00784 V=800.0 PL=0
MOVL C00785 V=800.0 PL=0
MOVL C00786 V=800.0 PL=0
MOVL C00787 V=800.0 PL=0
MOVL C00788 V=800.0 PL=0
MOVL C00789 V=800.0 PL=0
MOVL C00790 V=800.0 PL=0
MOVL C00791 V=800.0 PL=0
MOVL C00792 V=800.0 PL=0
MOVL C00793 V=800.0 PL=0
MOVL C00794 V=800.0 PL=0
MOVL C00795 V=800.0 PL=0
MOVL C00796 V=800.0 PL=0
MOVL C00797 V=800.0 PL=0
MOVL C00798 V=800.0 PL=0
MOVL C00799 V=800.0 PL=0
MOVL C00800 V=800.0 PL=0
MOVL C00801 V=800.0 PL=0
MOVL C00802 V=800.0 PL=0
MOVL C00803 V=800.0 PL=0
MOVL C00804 V=800.0 PL=0
MOVL C00805 V=800.0 PL=0
MOVL C00806 V=800.0 PL=0
MOVL C00807 V=800.0 PL=0
MOVL C00808 V=800.0 PL=0
MOVL C00809 V=800.0 PL=0
MOVL C00810 V=800.0 PL=0
MOVL C00811 V=800.0 PL=0
MOVL C00812 V=800.0 PL=0
MOVL C00813 V=800.0 PL=0
MOVL C00814 V=800.0 PL=0
MOVL C00815 V=800.0 PL=0
MOVL C00816 V=800.0 PL=0
MOVL C00817 V=800.0 PL=0
MOVL C00818 V=800.0 PL=0
MOVL C00819 V=800.0 PL=0
MOVL C00820 V=800.0 PL=0
MOVL C00821 V=800.0 PL=0
MOVL C00822 V=800.0 PL=0
MOVL C00823 V=800.0 PL=0
MOVL C00824 V=800.0 PL=0
MOVL C00825 V=800.0 PL=0
MOVL C00826 V=800.0 PL=0
MOVL C00827 V=800.0 PL=0
MOVL C00828 V=800.0 PL=0
MOVL C00829 V=800.0 PL=0
MOVL C00830 V=800.0 PL=0
MOVL C00831 V=800.0 PL=0
MOVL C00832 V=800.0 PL=0
MOVL C00833 V=800.0 PL=0
MOVL C00834 V=800.0 PL=0
MOVL C00835 V=800.0 PL=0
MOVL C00836 V=800.0 PL=0
MOVL C00837 V=800.0 PL=0
MOVL C00838 V=800.0 PL=0
MOVL C00839 V=800.0 PL=0
MOVL C00840 V=800.0 PL=0
MOVL C00841 V=800.0 PL=0
MOVL C00842 V=800.0 PL=0
MOVL C00843 V=800.0 PL=0
MOVL C00844 V=800.0 PL=0
MOVL C00845 V=800.0 PL=0
MOVL C00846 V=800.0 PL=0
MOVL C00847 V=800.0 PL=0
MOVL C00848 V=800.0 PL=0
MOVL C00849 V=800.0 PL=0
MOVL C00850 V=800.0 PL=0
MOVL C00851 V=800.0 PL=0
MOVL C00852 V=800.0 PL=0
MOVL C00853 V=800.0 PL=0
MOVL C00854 V=800.0 PL=0
MOVL C00855 V=800.0 PL=0
MOVL C00856 V=800.0 PL=0
MOVL C00857 V=800.0 PL=0
MOVL C00858 V=800.0 PL=0
MOVL C00859 V=800.0 PL=0
MOVL C00860 V=800.0 PL=0
MOVL C00861 V=800.0 PL=0
MOVL C00862 V=800.0 PL=0
MOVL C00863 V=800.0 PL=0
MOVL C00864 V=800.0 PL=0
MOVL C00865 V=800.0 PL=0
MOVL C00866 V=800.0 PL=0
MOVL C00867 V=800.0 PL=0
MOVL C00868 V=800.0 PL=0
MOVL C00869 V=800.0 PL=0
MOVL C00870 V=800.0 PL=0
MOVL C00871 V=800.0 PL=0
MOVL C00872 V=800.0 PL=0
MOVL C00873 V=800.0 PL=0
MOVL C00874 V=800.0 PL=0
MOVL C00875 V=800.0 PL=0
MOVL C00876 V=800.0 PL=0
MOVL C00877 V=800.0 PL=0
MOVL C00878 V=800.0 PL=0
MOVL C00879 V=800.0 PL=0
MOVL C00880 V=800.0 PL=0
MOVL C00881 V=800.0 PL=0
MOVL C00882 V=800.0 PL=0
MOVL C00883 V=800.0 PL=0
MOVL C00884 V=800.0 PL=0
MOVL C00885 V=800.0 PL=0
MOVL C00886 V=800.0 PL=0
MOVL C00887 V=800.0 PL=0
MOVL C00888 V=800.0 PL=0
MOVL C00889 V=800.0 PL=0
MOVL C00890 V=800.0 PL=0
MOVL C00891 V=800.0 PL=0
MOVL C00892 V=800.0 PL=0
MOVL C00893 V=800.0 PL=0
MOVL C00894 V=800.0 PL=0
MOVL C00895 V=800.0 PL=0
MOVL C00896 V=800.0 PL=0
MOVL C00897 V=800.0 PL=0
MOVL C00898 V=800.0 PL=0
MOVL C00899 V=800.0 PL=0
MOVL C00900 V=800.0 PL=0
MOVL C00901 V=800.0 PL=0
MOVL C00902 V=800.0 PL=0
MOVL C00903 V=800.0 PL=0
MOVL C00904 V=800.0 PL=0
MOVL C00905 V=800.0 PL=0
MOVL C00906 V=800.0 PL=0
MOVL C00907 V=800.0 PL=0
MOVL C00908 V=800.0 PL=0
MOVL C00909 V=800.0 PL=0
MOVL C00910 V=800.0 PL=0
MOVL C00911 V=800.0 PL=0
MOVL C00912 V=800.0 PL=0
MOVL C00913 V=800.0 PL=0
MOVL C00914 V=800.0 PL=0
MOVL C00915 V=800.0 PL=0
MOVL C00916 V=800.0 PL=0
MOVL C00917 V=800.0 PL=0
MOVL C00918 V=800.0 PL=0
MOVL C00919 V=800.0 PL=0
MOVL C00920 V=800.0 PL=0
MOVL C00921 V=800.0 PL=0
MOVL C00922 V=800.0 PL=0
MOVL C00923 V=800.0 PL=0
MOVL C00924 V=800.0 PL=0
MOVL C00925 V=800.0 PL=0
MOVL C00926 V=800.0 PL=0
MOVL C00927 V=800.0 PL=0
MOVL C00928 V=800.0 PL=0
MOVL C00929 V=800.0 PL=0
MOVL C00930 V=800.0 PL=0
MOVL C00931 V=800.0 PL=0
MOVL C00932 V=800.0 PL=0
MOVL C00933 V=800.0 PL=0
MOVL C00934 V=800.0 PL=0
MOVL C00935 V=800.0 PL=0
MOVL C00936 V=800.0 PL=0
MOVL C00937 V=800.0 PL=0
MOVL C00938 V=800.0 PL=0
MOVL C00939 V=800.0 PL=0
MOVL C00940 V=800.0 PL=0
MOVL C00941 V=800.0 PL=0
MOVL C00942 V=800.0 PL=0
MOVL C00943 V=800.0 PL=0
MOVL C00944 V=800.0 PL=0
MOVL C00945 V=800.0 PL=0
MOVL C00946 V=800.0 PL=0
MOVL C00947 V=800.0 PL=0
MOVL C00948 V=800.0 PL=0
MOVL C00949 V=800.0 PL=0
MOVL C00950 V=800.0 PL=0
MOVL C00951 V=800.0 PL=0
MOVL C00952 V=800.0 PL=0
MOVL C00953 V=800.0 PL=0
MOVL C00954 V=800.0 PL=0
MOVL C00955 V=800.0 PL=0
MOVL C00956 V=800.0 PL=0
MOVL C00957 V=800.0 PL=0
MOVL C00958 V=800.0 PL=0
MOVL C00959 V=800.0 PL=0
MOVL C00960 V=800.0 PL=0
MOVL C00961 V=800.0 PL=0
MOVL C00962 V=800.0 PL=0
MOVL C00963 V=800.0 PL=0
MOVL C00964 V=800.0 PL=0
MOVL C00965 V=800.0 PL=0
MOVL C00966 V=800.0 PL=0
MOVL C00967 V=800.0 PL=0
MOVL C00968 V=800.0 PL=0
MOVL C00969 V=800.0 PL=0
MOVL C00970 V=800.0 PL=0
MOVL C00971 V=800.0 PL=0
MOVL C00972 V=800.0 PL=0
MOVL C00973 V=800.0 PL=0
MOVL C00974 V=800.0 PL=0
MOVL C00975 V=800.0 PL=0
MOVL C00976 V=800.0 PL=0
MOVL C00977 V=800.0 PL=0
MOVL C00978 V=800.0 PL=0
MOVL C00979 V=800.0 PL=0
MOVL C00980 V=800.0 PL=0
MOVL C00981 V=800.0 PL=0
MOVL C00982 V=800.0 PL=0
MOVL C00983 V=800.0 PL=0
MOVL C00984 V=800.0 PL=0
MOVL C00985 V=800.0 PL=0
MOVL C00986 V=800.0 PL=0
MOVL C00987 V=800.0 PL=0
MOVL C00988 V=800.0 PL=0
MOVL C00989 V=800.0 PL=0
MOVL C00990 V=800.0 PL=0
MOVL C00991 V=800.0 PL=0
MOVL C00992 V=800.0 PL=0
MOVL C00993 V=800.0 PL=0
MOVL C00994 V=800.0 PL=0
MOVL C00995 V=800.0 PL=0
MOVL C00996 V=800.0 PL=0
MOVL C00997 V=800.0 PL=0
MOVL C00998 V=800.0 PL=0
MOVL C00999 V=800.0 PL=0
MOVL C01000 V=800.0 PL=0
MOVL C01001 V=800.0 PL=0
MOVL C01002 V=800.0 PL=0
MOVL C01003 V=800.0 PL=0
MOVL C01004 V=800.0 PL=0
MOVL C01005 V=800.0 PL=0
MOVL C01006 V=800.0 PL=0
MOVL C01007 V=800.0 PL=0
MOVL C01008 V=800.0 PL=0
MOVL C01009 V=800.0 PL=0
MOVL C01010 V=800.0 PL=0
MOVL C01011 V=800.0 PL=0
MOVL C01012 V=800.0 PL=0
MOVL C01013 V=800.0 PL=0
MOVL C01014 V=800.0 PL=0
MOVL C01015 V=800.0 PL=0
MOVL C01016 V=800.0 PL=0
MOVL C01017 V=800.0 PL=0
MOVL C01018 V=800.0 PL=0
MOVL C01019 V=800.0 PL=0
MOVL C01020 V=800.0 PL=0
MOVL C01021 V=800.0 PL=0
MOVL C01022 V=800.0 PL=0
MOVL C01023 V=800.0 PL=0
MOVL C01024 V=800.0 PL=0
MOVL C01025 V=800.0 PL=0
MOVL C01026 V=800.0 PL=0
MOVL C01027 V=800.0 PL=0
MOVL C01028 V=800.0 PL=0
MOVL C01029 V=800.0 PL=0
MOVL C01030 V=800.0 PL=0
MOVL C01031 V=800.0 PL=0
MOVL C01032 V=800.0 PL=0
MOVL C01033 V=800.0 PL=0
MOVL C01034 V=800.0 PL=0
MOVL C01035 V=800.0 PL=0
MOVL C01036 V=800.0 PL=0
MOVL C01037 V=800.0 PL=0
MOVL C01038 V=800.0 PL=0
MOVL C01039 V=800.0 PL=0
MOVL C01040 V=800.0 PL=0
MOVL C01041 V=800.0 PL=0
MOVL C01042 V=800.0 PL=0
MOVL C01043 V=800.0 PL=0
MOVL C01044 V=800.0 PL=0
MOVL C01045 V=800.0 PL=0
MOVL C01046 V=800.0 PL=0
MOVL C01047 V=800.0 PL=0
MOVL C01048 V=800.0 PL=0
MOVL C01049 V=800.0 PL=0
MOVL C01050 V=800.0 PL=0
MOVL C01051 V=800.0 PL=0
MOVL C01052 V=800.0 PL=0
MOVL C01053 V=800.0 PL=0
MOVL C01054 V=800.0 PL=0
MOVL C01055 V=800.0 PL=0
MOVL C01056 V=800.0 PL=0
MOVL C01057 V=800.0 PL=0
MOVL C01058 V=800.0 PL=0
MOVL C01059 V=800.0 PL=0
MOVL C01060 V=800.0 PL=0
MOVL C01061 V=800.0 PL=0
MOVL C01062 V=800.0 PL=0
MOVL C01063 V=800.0 PL=0
MOVL C01064 V=800.0 PL=0
MOVL C01065 V=800.0 PL=0
MOVL C01066 V=800.0 PL=0
MOVL C01067 V=800.0 PL=0
MOVL C01068 V=800.0 PL=0
MOVL C01069 V=800.0 PL=0
MOVL C01070 V=800.0 PL=0
MOVL C01071 V=800.0 PL=0
MOVL C01072 V=800.0 PL=0
MOVL C01073 V=800.0 PL=0
MOVL C01074 V=800.0 PL=0
MOVL C01075 V=800.0 PL=0
MOVL C01076 V=800.0 PL=0
MOVL C01077 V=800.0 PL=0
MOVL C01078 V=800.0 PL=0
MOVL C01079 V=800.0 PL=0
MOVL C01080 V=800.0 PL=0
MOVL C01081 V=800.0 PL=0
MOVL C01082 V=800.0 PL=0
MOVL C01083 V=800.0 PL=0
MOVL C01084 V=800.0 PL=0
MOVL C01085 V=800.0 PL=0
MOVL C01086 V=800.0 PL=0
MOVL C01087 V=800.0 PL=0
MOVL C01088 V=800.0 PL=0
MOVL C01089 V=800.0 PL=0
MOVL C01090 V=800.0 PL=0
MOVL C01091 V=800.0 PL=0
MOVL C01092 V=800.0 PL=0
MOVL C01093 V=800.0 PL=0
MOVL C01094 V=800.0 PL=0
MOVL C01095 V=800.0 PL=0
MOVL C01096 V=800.0 PL=0
MOVL C01097 V=800.0 PL=0
MOVL C01098 V=800.0 PL=0
MOVL C01099 V=800.0 PL=0
MOVL C01100 V=800.0 PL=0
MOVL C01101 V=800.0 PL=0
MOVL C01102 V=800.0 PL=0
MOVL C01103 V=800.0 PL=0
MOVL C01104 V=800.0 PL=0
MOVL C01105 V=800.0 PL=0
MOVL C01106 V=800.0 PL=0
MOVL C01107 V=800.0 PL=0
MOVL C01108 V=800.0 PL=0
MOVL C01109 V=800.0 PL=0
MOVL C01110 V=800.0 PL=0
MOVL C01111 V=800.0 PL=0
MOVL C01112 V=800.0 PL=0
MOVL C01113 V=800.0 PL=0
MOVL C01114 V=800.0 PL=0
MOVL C01115 V=800.0 PL=0
MOVL C01116 V=800.0 PL=0
MOVL C01117 V=800.0 PL=0
MOVL C01118 V=800.0 PL=0
MOVL C01119 V=800.0 PL=0
MOVL C01120 V=800.0 PL=0
MOVL C01121 V=800.0 PL=0
MOVL C01122 V=800.0 PL=0
MOVL C01123 V=800.0 PL=0
MOVL C01124 V=800.0 PL=0
MOVL C01125 V=800.0 PL=0
MOVL C01126 V=800.0 PL=0
MOVL C01127 V=800.0 PL=0
MOVL C01128 V=800.0 PL=0
MOVL C01129 V=800.0 PL=0
MOVL C01130 V=800.0 PL=0
MOVL C01131 V=800.0 PL=0
MOVL C01132 V=800.0 PL=0
MOVL C01133 V=800.0 PL=0
MOVL C01134 V=800.0 PL=0
MOVL C01135 V=800.0 PL=0
MOVL C01136 V=800.0 PL=0
MOVL C01137 V=800.0 PL=0
MOVL C01138 V=800.0 PL=0
MOVL C01139 V=800.0 PL=0
MOVL C01140 V=800.0 PL=0
MOVL C01141 V=800.0 PL=0
MOVL C01142 V=800.0 PL=0
MOVL C01143 V=800.0 PL=0
MOVL C01144 V=800.0 PL=0
MOVL C01145 V=800.0 PL=0
MOVL C01146 V=800.0 PL=0
MOVL C01147 V=800.0 PL=0
MOVL C01148 V=800.0 PL=0
MOVL C01149 V=800.0 PL=0
MOVL C01150 V=800.0 PL=0
MOVL C01151 V=800.0 PL=0
MOVL C01152 V=800.0 PL=0
MOVL C01153 V=800.0 PL=0
MOVL C01154 V=800.0 PL=0
MOVL C01155 V=800.0 PL=0
MOVL C01156 V=800.0 PL=0
MOVL C01157 V=800.0 PL=0
MOVL C01158 V=800.0 PL=0
MOVL C01159 V=800.0 PL=0
MOVL C01160 V=800.0 PL=0
MOVL C01161 V=800.0 PL=0
MOVL C01162 V=800.0 PL=0
MOVL C01163 V=800.0 PL=0
MOVL C01164 V=800.0 PL=0
MOVL C01165 V=800.0 PL=0
MOVL C01166 V=800.0 PL=0
MOVL C01167 V=800.0 PL=0
MOVL C01168 V=800.0 PL=0
MOVL C01169 V=800.0 PL=0
MOVL C01170 V=800.0 PL=0
MOVL C01171 V=800.0 PL=0
MOVL C01172 V=800.0 PL=0
MOVL C01173 V=800.0 PL=0
MOVL C01174 V=800.0 PL=0
MOVL C01175 V=800.0 PL=0
MOVL C01176 V=800.0 PL=0
MOVL C01177 V=800.0 PL=0
MOVL C01178 V=800.0 PL=0
MOVL C01179 V=800.0 PL=0
MOVL C01180 V=800.0 PL=0
MOVL C01181 V=800.0 PL=0
MOVL C01182 V=800.0 PL=0
MOVL C01183 V=800.0 PL=0
MOVL C01184 V=800.0 PL=0
MOVL C01185 V=800.0 PL=0
MOVL C01186 V=800.0 PL=0
MOVL C01187 V=800.0 PL=0
MOVL C01188 V=800.0 PL=0
MOVL C01189 V=800.0 PL=0
MOVL C01190 V=800.0 PL=0
MOVL C01191 V=800.0 PL=0
MOVL C01192 V=800.0 PL=0
MOVL C01193 V=800.0 PL=0
MOVL C01194 V=800.0 PL=0
MOVL C01195 V=800.0 PL=0
MOVL C01196 V=800.0 PL=0
MOVL C01197 V=800.0 PL=0
MOVL C01198 V=800.0 PL=0
MOVL C01199 V=800.0 PL=0
MOVL C01200 V=800.0 PL=0
MOVL C01201 V=800.0 PL=0
MOVL C01202 V=800.0 PL=0
MOVL C01203 V=800.0 PL=0
MOVL C01204 V=800.0 PL=0
MOVL C01205 V=800.0 PL=0
MOVL C01206 V=800.0 PL=0
MOVL C01207 V=800.0 PL=0
MOVL C01208 V=800.0 PL=0
MOVL C01209 V=800.0 PL=0
MOVL C01210 V=800.0 PL=0
MOVL C01211 V=800.0 PL=0
MOVL C01212 V=800.0 PL=0
MOVL C01213 V=800.0 PL=0
MOVL C01214 V=800.0 PL=0
MOVL C01215 V=800.0 PL=0
MOVL C01216 V=800.0 PL=0
MOVL C01217 V=800.0 PL=0
MOVL C01218 V=800.0 PL=0
MOVL C01219 V=800.0 PL=0
MOVL C01220 V=800.0 PL=0
MOVL C01221 V=800.0 PL=0
MOVL C01222 V=800.0 PL=0
MOVL C01223 V=800.0 PL=0
MOVL C01224 V=800.0 PL=0
MOVL C01225 V=800.0 PL=0
MOVL C01226 V=800.0 PL=0
MOVL C01227 V=800.0 PL=0
MOVL C01228 V=800.0 PL=0
MOVL C01229 V=800.0 PL=0
MOVL C01230 V=800.0 PL=0
MOVL C01231 V=800.0 PL=0
MOVL C01232 V=800.0 PL=0
MOVL C01233 V=800.0 PL=0
MOVL C01234 V=800.0 PL=0
MOVL C01235 V=800.0 PL=0
MOVL C01236 V=800.0 PL=0
MOVL C01237 V=800.0 PL=0
MOVL C01238 V=800.0 PL=0
MOVL C01239 V=800.0 PL=0
MOVL C01240 V=800.0 PL=0
MOVL C01241 V=800.0 PL=0
MOVL C01242 V=800.0 PL=0
MOVL C01243 V=800.0 PL=0
MOVL C01244 V=800.0 PL=0
MOVL C01245 V=800.0 PL=0
MOVL C01246 V=800.0 PL=0
MOVL C01247 V=800.0 PL=0
MOVL C01248 V=800.0 PL=0
MOVL C01249 V=800.0 PL=0
MOVL C01250 V=800.0 PL=0
MOVL C01251 V=800.0 PL=0
MOVL C01252 V=800.0 PL=0
MOVL C01253 V=800.0 PL=0
MOVL C01254 V=800.0 PL=0
MOVL C01255 V=800.0 PL=0
MOVL C01256 V=800.0 PL=0
MOVL C01257 V=800.0 PL=0
MOVL C01258 V=800.0 PL=0
MOVL C01259 V=800.0 PL=0
MOVL C01260 V=800.0 PL=0
MOVL C01261 V=800.0 PL=0
MOVL C01262 V=800.0 PL=0
MOVL C01263 V=800.0 PL=0
MOVL C01264 V=800.0 PL=0
MOVL C01265 V=800.0 PL=0
MOVL C01266 V=800.0 PL=0
MOVL C01267 V=800.0 PL=0
MOVL C01268 V=800.0 PL=0
MOVL C01269 V=800.0 PL=0
MOVL C01270 V=800.0 PL=0
MOVL C01271 V=800.0 PL=0
MOVL C01272 V=800.0 PL=0
MOVL C01273 V=800.0 PL=0
MOVL C01274 V=800.0 PL=0
MOVL C01275 V=800.0 PL=0
MOVL C01276 V=800.0 PL=0
MOVL C01277 V=800.0 PL=0
MOVL C01278 V=800.0 PL=0
MOVL C01279 V=800.0 PL=0
MOVL C01280 V=800.0 PL=0
MOVL C01281 V=800.0 PL=0
MOVL C01282 V=800.0 PL=0
MOVL C01283 V=800.0 PL=0
MOVL C01284 V=800.0 PL=0
MOVL C01285 V=800.0 PL=0
MOVL C01286 V=800.0 PL=0
MOVL C01287 V=800.0 PL=0
MOVL C01288 V=800.0 PL=0
MOVL C01289 V=800.0 PL=0
MOVL C01290 V=800.0 PL=0
MOVL C01291 V=800.0 PL=0
MOVL C01292 V=800.0 PL=0
MOVL C01293 V=800.0 PL=0
MOVL C01294 V=800.0 PL=0
MOVL C01295 V=800.0 PL=0
MOVL C01296 V=800.0 PL=0
MOVL C01297 V=800.0 PL=0
MOVL C01298 V=800.0 PL=0
MOVL C01299 V=800.0 PL=0
MOVL C01300 V=800.0 PL=0
MOVL C01301 V=800.0 PL=0
MOVL C01302 V=800.0 PL=0
MOVL C01303 V=800.0 PL=0
MOVL C01304 V=800.0 PL=0
MOVL C01305 V=800.0 PL=0
MOVL C01306 V=800.0 PL=0
MOVL C01307 V=800.0 PL=0
MOVL C01308 V=800.0 PL=0
MOVL C01309 V=800.0 PL=0
MOVL C01310 V=800.0 PL=0
MOVL C01311 V=800.0 PL=0
MOVL C01312 V=800.0 PL=0
MOVL C01313 V=800.0 PL=0
MOVL C01314 V=800.0 PL=0
MOVL C01315 V=800.0 PL=0
MOVL C01316 V=800.0 PL=0
MOVL C01317 V=800.0 PL=0
MOVL C01318 V=800.0 PL=0
MOVL C01319 V=800.0 PL=0
MOVL C01320 V=800.0 PL=0
MOVL C01321 V=800.0 PL=0
MOVL C01322 V=800.0 PL=0
MOVL C01323 V=800.0 PL=0
MOVL C01324 V=800.0 PL=0
MOVL C01325 V=800.0 PL=0
MOVL C01326 V=800.0 PL=0
MOVL C01327 V=800.0 PL=0
MOVL C01328 V=800.0 PL=0
MOVL C01329 V=800.0 PL=0
MOVL C01330 V=800.0 PL=0
MOVL C01331 V=800.0 PL=0
MOVL C01332 V=800.0 PL=0
MOVL C01333 V=800.0 PL=0
MOVL C01334 V=800.0 PL=0
MOVL C01335 V=800.0 PL=0
MOVL C01336 V=800.0 PL=0
MOVL C01337 V=800.0 PL=0
MOVL C01338 V=800.0 PL=0
MOVL C01339 V=800.0 PL=0
MOVL C01340 V=800.0 PL=0
MOVL C01341 V=800.0 PL=0
MOVL C01342 V=800.0 PL=0
MOVL C01343 V=800.0 PL=0
MOVL C01344 V=800.0 PL=0
MOVL C01345 V=800.0 PL=0
MOVL C01346 V=800.0 PL=0
MOVL C01347 V=800.0 PL=0
MOVL C01348 V=800.0 PL=0
MOVL C01349 V=800.0 PL=0
MOVL C01350 V=800.0 PL=0
MOVL C01351 V=800.0 PL=0
MOVL C01352 V=800.0 PL=0
MOVL C01353 V=800.0 PL=0
MOVL C01354 V=800.0 PL=0
MOVL C01355 V=800.0 PL=0
MOVL C01356 V=800.0 PL=0
MOVL C01357 V=800.0 PL=0
MOVL C01358 V=800.0 PL=0
MOVL C01359 V=800.0 PL=0
MOVL C01360 V=800.0 PL=0
MOVL C01361 V=800.0 PL=0
MOVL C01362 V=800.0 PL=0
MOVL C01363 V=800.0 PL=0
MOVL C01364 V=800.0 PL=0
MOVL C01365 V=800.0 PL=0
MOVL C01366 V=800.0 PL=0
MOVL C01367 V=800.0 PL=0
MOVL C01368 V=800.0 PL=0
MOVL C01369 V=800.0 PL=0
MOVL C01370 V=800.0 PL=0
MOVL C01371 V=800.0 PL=0
MOVL C01372 V=800.0 PL=0
MOVL C01373 V=800.0 PL=0
MOVL C01374 V=800.0 PL=0
MOVL C01375 V=800.0 PL=0
MOVL C01376 V=800.0 PL=0
MOVL C01377 V=800.0 PL=0
MOVL C01378 V=800.0 PL=0
MOVL C01379 V=800.0 PL=0
MOVL C01380 V=800.0 PL=0
MOVL C01381 V=800.0 PL=0
MOVL C01382 V=800.0 PL=0
MOVL C01383 V=800.0 PL=0
MOVL C01384 V=800.0 PL=0
MOVL C01385 V=800.0 PL=0
MOVL C01386 V=800.0 PL=0
MOVL C01387 V=800.0 PL=0
MOVL C01388 V=800.0 PL=0
MOVL C01389 V=800.0 PL=0
MOVL C01390 V=800.0 PL=0
MOVL C01391 V=800.0 PL=0
MOVL C01392 V=800.0 PL=0
MOVL C01393 V=800.0 PL=0
MOVL C01394 V=800.0 PL=0
MOVL C01395 V=800.0 PL=0
MOVL C01396 V=800.0 PL=0
MOVL C01397 V=800.0 PL=0
MOVL C01398 V=800.0 PL=0
MOVL C01399 V=800.0 PL=0
MOVL C01400 V=800.0 PL=0
MOVL C01401 V=800.0 PL=0
MOVL C01402 V=800.0 PL=0
MOVL C01403 V=800.0 PL=0
MOVL C01404 V=800.0 PL=0
MOVL C01405 V=800.0 PL=0
MOVL C01406 V=800.0 PL=0
MOVL C01407 V=800.0 PL=0
MOVL C01408 V=800.0 PL=0
MOVL C01409 V=800.0 PL=0
MOVL C01410 V=800.0 PL=0
MOVL C01411 V=800.0 PL=0
MOVL C01412 V=800.0 PL=0
MOVL C01413 V=800.0 PL=0
MOVL C01414 V=800.0 PL=0
MOVL C01415 V=800.0 PL=0
MOVL C01416 V=800.0 PL=0
MOVL C01417 V=800.0 PL=0
MOVL C01418 V=800.0 PL=0
MOVL C01419 V=800.0 PL=0
MOVL C01420 V=800.0 PL=0
MOVL C01421 V=800.0 PL=0
MOVL C01422 V=800.0 PL=0
MOVL C01423 V=800.0 PL=0
MOVL C01424 V=800.0 PL=0
MOVL C01425 V=800.0 PL=0
MOVL C01426 V=800.0 PL=0
MOVL C01427 V=800.0 PL=0
MOVL C01428 V=800.0 PL=0
MOVL C01429 V=800.0 PL=0
MOVL C01430 V=800.0 PL=0
MOVL C01431 V=800.0 PL=0
MOVL C01432 V=800.0 PL=0
MOVL C01433 V=800.0 PL=0
MOVL C01434 V=800.0 PL=0
MOVL C01435 V=800.0 PL=0
MOVL C01436 V=800.0 PL=0
MOVL C01437 V=800.0 PL=0
MOVL C01438 V=800.0 PL=0
MOVL C01439 V=800.0 PL=0
MOVL C01440 V=800.0 PL=0
MOVL C01441 V=800.0 PL=0
MOVL C01442 V=800.0 PL=0
MOVL C01443 V=800.0 PL=0
MOVL C01444 V=800.0 PL=0
MOVL C01445 V=800.0 PL=0
MOVL C01446 V=800.0 PL=0
MOVL C01447 V=800.0 PL=0
MOVL C01448 V=800.0 PL=0
MOVL C01449 V=800.0 PL=0
MOVL C01450 V=800.0 PL=0
MOVL C01451 V=800.0 PL=0
MOVL C01452 V=800.0 PL=0
MOVL C01453 V=800.0 PL=0
MOVL C01454 V=800.0 PL=0
MOVL C01455 V=800.0 PL=0
MOVL C01456 V=800.0 PL=0
MOVL C01457 V=800.0 PL=0
MOVL C01458 V=800.0 PL=0
MOVL C01459 V=800.0 PL=0
MOVL C01460 V=800.0 PL=0
MOVL C01461 V=800.0 PL=0
MOVL C01462 V=800.0 PL=0
MOVL C01463 V=800.0 PL=0
MOVL C01464 V=800.0 PL=0
MOVL C01465 V=800.0 PL=0
MOVL C01466 V=800.0 PL=0
MOVL C01467 V=800.0 PL=0
MOVL C01468 V=800.0 PL=0
MOVL C01469 V=800.0 PL=0
MOVL C01470 V=800.0 PL=0
MOVL C01471 V=800.0 PL=0
MOVL C01472 V=800.0 PL=0
MOVL C01473 V=800.0 PL=0
MOVL C01474 V=800.0 PL=0
MOVL C01475 V=800.0 PL=0
MOVL C01476 V=800.0 PL=0
MOVL C01477 V=800.0 PL=0
MOVL C01478 V=800.0 PL=0
MOVL C01479 V=800.0 PL=0
MOVL C01480 V=800.0 PL=0
MOVL C01481 V=800.0 PL=0
MOVL C01482 V=800.0 PL=0
MOVL C01483 V=800.0 PL=0
MOVL C01484 V=800.0 PL=0
MOVL C01485 V=800.0 PL=0
MOVL C01486 V=800.0 PL=0
MOVL C01487 V=800.0 PL=0
MOVL C01488 V=800.0 PL=0
MOVL C01489 V=800.0 PL=0
MOVL C01490 V=800.0 PL=0
MOVL C01491 V=800.0 PL=0
MOVL C01492 V=800.0 PL=0
MOVL C01493 V=800.0 PL=0
MOVL C01494 V=800.0 PL=0
MOVL C01495 V=800.0 PL=0
MOVL C01496 V=800.0 PL=0
MOVL C01497 V=800.0 PL=0
MOVL C01498 V=800.0 PL=0
MOVL C01499 V=800.0 PL=0
MOVL C01500 V=800.0 PL=0
MOVL C01501 V=800.0 PL=0
MOVL C01502 V=800.0 PL=0
MOVL C01503 V=800.0 PL=0
MOVL C01504 V=800.0 PL=0
MOVL C01505 V=800.0 PL=0
MOVL C01506 V=800.0 PL=0
MOVL C01507 V=800.0 PL=0
MOVL C01508 V=800.0 PL=0
MOVL C01509 V=800.0 PL=0
MOVL C01510 V=800.0 PL=0
MOVL C01511 V=800.0 PL=0
MOVL C01512 V=800.0 PL=0
MOVL C01513 V=800.0 PL=0
MOVL C01514 V=800.0 PL=0
MOVL C01515 V=800.0 PL=0
MOVL C01516 V=800.0 PL=0
MOVL C01517 V=800.0 PL=0
MOVL C01518 V=800.0 PL=0
MOVL C01519 V=800.0 PL=0
MOVL C01520 V=800.0 PL=0
MOVL C01521 V=800.0 PL=0
MOVL C01522 V=800.0 PL=0
MOVL C01523 V=800.0 PL=0
MOVL C01524 V=800.0 PL=0
MOVL C01525 V=800.0 PL=0
MOVL C01526 V=800.0 PL=0
MOVL C01527 V=800.0 PL=0
MOVL C01528 V=800.0 PL=0
MOVL C01529 V=800.0 PL=0
MOVL C01530 V=800.0 PL=0
MOVL C01531 V=800.0 PL=0
MOVL C01532 V=800.0 PL=0
MOVL C01533 V=800.0 PL=0
MOVL C01534 V=800.0 PL=0
MOVL C01535 V=800.0 PL=0
MOVL C01536 V=800.0 PL=0
MOVL C01537 V=800.0 PL=0
MOVL C01538 V=800.0 PL=0
MOVL C01539 V=800.0 PL=0
MOVL C01540 V=800.0 PL=0
MOVL C01541 V=800.0 PL=0
MOVL C01542 V=800.0 PL=0
MOVL C01543 V=800.0 PL=0
MOVL C01544 V=800.0 PL=0
MOVL C01545 V=800.0 PL=0
MOVL C01546 V=800.0 PL=0
MOVL C01547 V=800.0 PL=0
MOVL C01548 V=800.0 PL=0
MOVL C01549 V=800.0 PL=0
MOVL C01550 V=800.0 PL=0
MOVL C01551 V=800.0 PL=0
MOVL C01552 V=800.0 PL=0
MOVL C01553 V=800.0 PL=0
MOVL C01554 V=800.0 PL=0
MOVL C01555 V=800.0 PL=0
MOVL C01556 V=800.0 PL=0
MOVL C01557 V=800.0 PL=0
MOVL C01558 V=800.0 PL=0
MOVL C01559 V=800.0 PL=0
MOVL C01560 V=800.0 PL=0
MOVL C01561 V=800.0 PL=0
MOVL C01562 V=800.0 PL=0
MOVL C01563 V=800.0 PL=0
MOVL C01564 V=800.0 PL=0
MOVL C01565 V=800.0 PL=0
MOVL C01566 V=800.0 PL=0
MOVL C01567 V=800.0 PL=0
MOVL C01568 V=800.0 PL=0
MOVL C01569 V=800.0 PL=0
MOVL C01570 V=800.0 PL=0
MOVL C01571 V=800.0 PL=0
MOVL C01572 V=800.0 PL=0
MOVL C01573 V=800.0 PL=0
MOVL C01574 V=800.0 PL=0
MOVL C01575 V=800.0 PL=0
MOVL C01576 V=800.0 PL=0
MOVL C01577 V=800.0 PL=0
MOVL C01578 V=800.0 PL=0
MOVL C01579 V=800.0 PL=0
MOVL C01580 V=800.0 PL=0
MOVL C01581 V=800.0 PL=0
MOVL C01582 V=800.0 PL=0
MOVL C01583 V=800.0 PL=0
MOVL C01584 V=800.0 PL=0
MOVL C01585 V=800.0 PL=0
MOVL C01586 V=800.0 PL=0
MOVL C01587 V=800.0 PL=0
MOVL C01588 V=800.0 PL=0
MOVL C01589 V=800.0 PL=0
MOVL C01590 V=800.0 PL=0
MOVL C01591 V=800.0 PL=0
MOVL C01592 V=800.0 PL=0
MOVL C01593 V=800.0 PL=0
MOVL C01594 V=800.0 PL=0
MOVL C01595 V=800.0 PL=0
MOVL C01596 V=800.0 PL=0
MOVL C01597 V=800.0 PL=0
MOVL C01598 V=800.0 PL=0
MOVL C01599 V=800.0 PL=0
MOVL C01600 V=800.0 PL=0
MOVL C01601 V=800.0 PL=0
MOVL C01602 V=800.0 PL=0
MOVL C01603 V=800.0 PL=0
MOVL C01604 V=800.0 PL=0
MOVL C01605 V=800.0 PL=0
MOVL C01606 V=800.0 PL=0
MOVL C01607 V=800.0 PL=0
MOVL C01608 V=800.0 PL=0
MOVL C01609 V=800.0 PL=0
MOVL C01610 V=800.0 PL=0
MOVL C01611 V=800.0 PL=0
MOVL C01612 V=800.0 PL=0
MOVL C01613 V=800.0 PL=0
MOVL C01614 V=800.0 PL=0
MOVL C01615 V=800.0 PL=0
MOVL C01616 V=800.0 PL=0
MOVL C01617 V=800.0 PL=0
MOVL C01618 V=800.0 PL=0
MOVL C01619 V=800.0 PL=0
MOVL C01620 V=800.0 PL=0
MOVL C01621 V=800.0 PL=0
MOVL C01622 V=800.0 PL=0
MOVL C01623 V=800.0 PL=0
MOVL C01624 V=800.0 PL=0
MOVL C01625 V=800.0 PL=0
MOVL C01626 V=800.0 PL=0
MOVL C01627 V=800.0 PL=0
MOVL C01628 V=800.0 PL=0
MOVL C01629 V=800.0 PL=0
MOVL C01630 V=800.0 PL=0
MOVL C01631 V=800.0 PL=0
MOVL C01632 V=800.0 PL=0
MOVL C01633 V=800.0 PL=0
MOVL C01634 V=800.0 PL=0
MOVL C01635 V=800.0 PL=0
MOVL C01636 V=800.0 PL=0
MOVL C01637 V=800.0 PL=0
MOVL C01638 V=800.0 PL=0
MOVL C01639 V=800.0 PL=0
MOVL C01640 V=800.0 PL=0
MOVL C01641 V=800.0 PL=0
MOVL C01642 V=800.0 PL=0
MOVL C01643 V=800.0 PL=0
MOVL C01644 V=800.0 PL=0
MOVL C01645 V=800.0 PL=0
MOVL C01646 V=800.0 PL=0
MOVL C01647 V=800.0 PL=0
MOVL C01648 V=800.0 PL=0
MOVL C01649 V=800.0 PL=0
MOVL C01650 V=800.0 PL=0
MOVL C01651 V=800.0 PL=0
MOVL C01652 V=800.0 PL=0
MOVL C01653 V=800.0 PL=0
MOVL C01654 V=800.0 PL=0
MOVL C01655 V=800.0 PL=0
MOVL C01656 V=800.0 PL=0
MOVL C01657 V=800.0 PL=0
MOVL C01658 V=800.0 PL=0
MOVL C01659 V=800.0 PL=0
MOVL C01660 V=800.0 PL=0
MOVL C01661 V=800.0 PL=0
MOVL C01662 V=800.0 PL=0
MOVL C01663 V=800.0 PL=0
MOVL C01664 V=800.0 PL=0
MOVL C01665 V=800.0 PL=0
MOVL C01666 V=800.0 PL=0
MOVL C01667 V=800.0 PL=0
MOVL C01668 V=800.0 PL=0
MOVL C01669 V=800.0 PL=0
MOVL C01670 V=800.0 PL=0
MOVL C01671 V=800.0 PL=0
MOVL C01672 V=800.0 PL=0
MOVL C01673 V=800.0 PL=0
MOVL C01674 V=800.0 PL=0
MOVL C01675 V=800.0 PL=0
MOVL C01676 V=800.0 PL=0
MOVL C01677 V=800.0 PL=0
MOVL C01678 V=800.0 PL=0
MOVL C01679 V=800.0 PL=0
MOVL C01680 V=800.0 PL=0
MOVL C01681 V=800.0 PL=0
MOVL C01682 V=800.0 PL=0
MOVL C01683 V=800.0 PL=0
MOVL C01684 V=800.0 PL=0
MOVL C01685 V=800.0 PL=0
MOVL C01686 V=800.0 PL=0
MOVL C01687 V=800.0 PL=0
MOVL C01688 V=800.0 PL=0
MOVL C01689 V=800.0 PL=0
MOVL C01690 V=800.0 PL=0
MOVL C01691 V=800.0 PL=0
MOVL C01692 V=800.0 PL=0
MOVL C01693 V=800.0 PL=0
MOVL C01694 V=800.0 PL=0
MOVL C01695 V=800.0 PL=0
MOVL C01696 V=800.0 PL=0
MOVL C01697 V=800.0 PL=0
MOVL C01698 V=800.0 PL=0
MOVL C01699 V=800.0 PL=0
MOVL C01700 V=800.0 PL=0
MOVL C01701 V=800.0 PL=0
MOVL C01702 V=800.0 PL=0
MOVL C01703 V=800.0 PL=0
MOVL C01704 V=800.0 PL=0
MOVL C01705 V=800.0 PL=0
MOVL C01706 V=800.0 PL=0
MOVL C01707 V=800.0 PL=0
MOVL C01708 V=800.0 PL=0
MOVL C01709 V=800.0 PL=0
MOVL C01710 V=800.0 PL=0
MOVL C01711 V=800.0 PL=0
MOVL C01712 V=800.0 PL=0
MOVL C01713 V=800.0 PL=0
MOVL C01714 V=800.0 PL=0
MOVL C01715 V=800.0 PL=0
MOVL C01716 V=800.0 PL=0
MOVL C01717 V=800.0 PL=0
MOVL C01718 V=800.0 PL=0
MOVL C01719 V=800.0 PL=0
MOVL C01720 V=800.0 PL=0
MOVL C01721 V=800.0 PL=0
MOVL C01722 V=800.0 PL=0
MOVL C01723 V=800.0 PL=0
MOVL C01724 V=800.0 PL=0
MOVL C01725 V=800.0 PL=0
MOVL C01726 V=800.0 PL=0
MOVL C01727 V=800.0 PL=0
MOVL C01728 V=800.0 PL=0
MOVL C01729 V=800.0 PL=0
MOVL C01730 V=800.0 PL=0
MOVL C01731 V=800.0 PL=0
MOVL C01732 V=800.0 PL=0
MOVL C01733 V=800.0 PL=0
MOVL C01734 V=800.0 PL=0
MOVL C01735 V=800.0 PL=0
MOVL C01736 V=800.0 PL=0
MOVL C01737 V=800.0 PL=0
MOVL C01738 V=800.0 PL=0
MOVL C01739 V=800.0 PL=0
MOVL C01740 V=800.0 PL=0
MOVL C01741 V=800.0 PL=0
MOVL C01742 V=800.0 PL=0
MOVL C01743 V=800.0 PL=0
MOVL C01744 V=800.0 PL=0
MOVL C01745 V=800.0 PL=0
MOVL C01746 V=800.0 PL=0
MOVL C01747 V=800.0 PL=0
MOVL C01748 V=800.0 PL=0
MOVL C01749 V=800.0 PL=0
MOVL C01750 V=800.0 PL=0
MOVL C01751 V=800.0 PL=0
MOVL C01752 V=800.0 PL=0
MOVL C01753 V=800.0 PL=0
MOVL C01754 V=800.0 PL=0
MOVL C01755 V=800.0 PL=0
MOVL C01756 V=800.0 PL=0
MOVL C01757 V=800.0 PL=0
MOVL C01758 V=800.0 PL=0
MOVL C01759 V=800.0 PL=0
MOVL C01760 V=800.0 PL=0
MOVL C01761 V=800.0 PL=0
MOVL C01762 V=800.0 PL=0
MOVL C01763 V=800.0 PL=0
MOVL C01764 V=800.0 PL=0
MOVL C01765 V=800.0 PL=0
MOVL C01766 V=800.0 PL=0
MOVL C01767 V=800.0 PL=0
MOVL C01768 V=800.0 PL=0
MOVL C01769 V=800.0 PL=0
MOVL C01770 V=800.0 PL=0
MOVL C01771 V=800.0 PL=0
MOVL C01772 V=800.0 PL=0
MOVL C01773 V=800.0 PL=0
MOVL C01774 V=800.0 PL=0
MOVL C01775 V=800.0 PL=0
MOVL C01776 V=800.0 PL=0
MOVL C01777 V=800.0 PL=0
MOVL C01778 V=800.0 PL=0
MOVL C01779 V=800.0 PL=0
MOVL C01780 V=800.0 PL=0
MOVL C01781 V=800.0 PL=0
MOVL C01782 V=800.0 PL=0
MOVL C01783 V=800.0 PL=0
MOVL C01784 V=800.0 PL=0
MOVL C01785 V=800.0 PL=0
MOVL C01786 V=800.0 PL=0
MOVL C01787 V=800.0 PL=0
MOVL C01788 V=800.0 PL=0
MOVL C01789 V=800.0 PL=0
MOVL C01790 V=800.0 PL=0
MOVL C01791 V=800.0 PL=0
MOVL C01792 V=800.0 PL=0
MOVL C01793 V=800.0 PL=0
MOVL C01794 V=800.0 PL=0
MOVL C01795 V=800.0 PL=0
MOVL C01796 V=800.0 PL=0
